LIN {X 0,Y 177.119,Z 453.02,A -85,B 0,C 180,E1 -22409.999,E2 -22409.999} C_VEL
LIN {X 0,Y 176.439,Z 454.874,A -85,B 0,C 180,E1 -22414.569,E2 -22414.569} C_VEL
LIN {X 0,Y 176.286,Z 455.203,A -85,B 0,C 180,E1 -22416.868,E2 -22416.868} C_VEL
LIN {X 0,Y 176.801,Z 454.648,A -85,B 0,C 180,E1 -22421.463,E2 -22421.463} C_VEL
LIN {X 0,Y 178.406,Z 452.583,A -85,B 0,C 180,E1 -22426.006,E2 -22426.006} C_VEL
LIN {X 0,Y 180.457,Z 449.998,A -85,B 0,C 180,E1 -22429.331,E2 -22429.331} C_VEL
LIN {X 0,Y 183.132,Z 446.482,A -85,B 0,C 180,E1 -22432.567,E2 -22432.567} C_VEL
LIN {X 0,Y 186.346,Z 441.993,A -85,B 0,C 180,E1 -22435.703,E2 -22435.703} C_VEL
LIN {X 0,Y 191.105,Z 435.334,A -85,B 0,C 180,E1 -22439.161,E2 -22439.161} C_VEL
LIN {X 0,Y 195.82,Z 428.208,A -85,B 0,C 180,E1 -22441.963,E2 -22441.963} C_VEL
LIN {X 0,Y 201.029,Z 419.477,A -85,B 0,C 180,E1 -22444.617,E2 -22444.617} C_VEL
LIN {X 0,Y 205.808,Z 410.713,A -85,B 0,C 180,E1 -22446.697,E2 -22446.697} C_VEL
LIN {X 0,Y 210.975,Z 400.084,A -85,B 0,C 180,E1 -22448.652,E2 -22448.652} C_VEL
LIN {X 0,Y 215.413,Z 389.657,A -85,B 0,C 180,E1 -22450.117,E2 -22450.117} C_VEL
LIN {X 0,Y 219.48,Z 378.312,A -85,B 0,C 180,E1 -22451.333,E2 -22451.333} C_VEL
LIN {X 0,Y 223.276,Z 364.778,A -85,B 0,C 180,E1 -22452.437,E2 -22452.437} C_VEL
LIN {X 0,Y 226.064,Z 351.459,A -85,B 0,C 180,E1 -22453.198,E2 -22453.198} C_VEL
LIN {X 0,Y 228.603,Z 331.076,A -85,B 0,C 180,E1 -22453.998,E2 -22453.998} C_VEL
LIN {X 0,Y 229.847,Z 318.937,A -85,B 0,C 180,E1 -22454.478,E2 -22454.478} C_VEL
LIN {X 0,Y 229.863,Z 308.216,A -85,B 0,C 180,E1 -22455.412,E2 -22455.412} C_VEL
LIN {X 0,Y 227.63,Z 301.276,A -85,B 0,C 180,E1 -22457.167,E2 -22457.167} C_VEL
LIN {X 0,Y 225.204,Z 295.085,A -85,B 0,C 180,E1 -22459.217,E2 -22459.217} C_VEL
LIN {X 0,Y 223.459,Z 290.853,A -85,B 0,C 180,E1 -22460.87,E2 -22460.87} C_VEL
LIN {X 0,Y 221.449,Z 286.067,A -85,B 0,C 180,E1 -22463.095,E2 -22463.095} C_VEL
LIN {X 0,Y 219.336,Z 281.128,A -85,B 0,C 180,E1 -22466.096,E2 -22466.096} C_VEL
LIN {X 0,Y 217.144,Z 276.417,A -85,B 0,C 180,E1 -22471.174,E2 -22471.174} C_VEL
LIN {X 0,Y 216.832,Z 274.973,A -85,B 0,C 180,E1 -22475.167,E2 -22475.167} C_VEL
LIN {X 0,Y 217.513,Z 275.061,A -85,B 0,C 180,E1 -22478.561,E2 -22478.561} C_VEL
LIN {X 0,Y 218.482,Z 275.796,A -85,B 0,C 180,E1 -22480.742,E2 -22480.742} C_VEL
LIN {X 0,Y 220.281,Z 278.676,A -85,B 0,C 180,E1 -22483.828,E2 -22483.828} C_VEL
LIN {X 0,Y 221.098,Z 279.677,A -85,B 0,C 180,E1 -22484.873,E2 -22484.873} C_VEL
LIN {X 0,Y 223.871,Z 284.056,A -85,B 0,C 180,E1 -22487.867,E2 -22487.867} C_VEL
LIN {X 0,Y 226.551,Z 288.873,A -85,B 0,C 180,E1 -22490.248,E2 -22490.248} C_VEL
LIN {X 0,Y 229.149,Z 293.131,A -85,B 0,C 180,E1 -22492.167,E2 -22492.167} C_VEL
LIN {X 0,Y 231.689,Z 298.864,A -85,B 0,C 180,E1 -22493.945,E2 -22493.945} C_VEL
LIN {X 0,Y 227.767,Z 334.024,A -85,B 0,C 180,E1 -22495.35,E2 -22495.35} C_VEL
LIN {X 0,Y 225.731,Z 345.822,A -85,B 0,C 180,E1 -22496.11,E2 -22496.11} C_VEL
LIN {X 0,Y 222.631,Z 358.855,A -85,B 0,C 180,E1 -22497.286,E2 -22497.286} C_VEL
LIN {X 0,Y 218.74,Z 371.166,A -85,B 0,C 180,E1 -22498.758,E2 -22498.758} C_VEL
LIN {X 0,Y 214.991,Z 380.89,A -85,B 0,C 180,E1 -22500.234,E2 -22500.234} C_VEL
LIN {X 0,Y 210.962,Z 389.896,A -85,B 0,C 180,E1 -22501.957,E2 -22501.957} C_VEL
LIN {X 0,Y 205.904,Z 399.515,A -85,B 0,C 180,E1 -22504.288,E2 -22504.288} C_VEL
LIN {X 0,Y 200.682,Z 408.153,A -85,B 0,C 180,E1 -22507.04,E2 -22507.04} C_VEL
LIN {X 0,Y 196.113,Z 414.843,A -85,B 0,C 180,E1 -22509.8,E2 -22509.8} C_VEL
LIN {X 0,Y 192.012,Z 420.181,A -85,B 0,C 180,E1 -22512.686,E2 -22512.686} C_VEL
LIN {X 0,Y 187.629,Z 425.077,A -85,B 0,C 180,E1 -22516.315,E2 -22516.315} C_VEL
LIN {X 0,Y 183.961,Z 428.518,A -85,B 0,C 180,E1 -22520.11,E2 -22520.11} C_VEL
LIN {X 0,Y 181.959,Z 430.045,A -85,B 0,C 180,E1 -22522.721,E2 -22522.721} C_VEL
LIN {X 0,Y 179.89,Z 431.131,A -85,B 0,C 180,E1 -22526.03,E2 -22526.03} C_VEL
LIN {X 0,Y 178.152,Z 431.262,A -85,B 0,C 180,E1 -22529.787,E2 -22529.787} C_VEL
LIN {X 0,Y 176.979,Z 430.196,A -85,B 0,C 180,E1 -22533.776,E2 -22533.776} C_VEL
LIN {X 0,Y 176.467,Z 428.319,A -85,B 0,C 180,E1 -22537.201,E2 -22537.201} C_VEL
LIN {X 0,Y 176.435,Z 425.306,A -85,B 0,C 180,E1 -22540.815,E2 -22540.815} C_VEL
LIN {X 0,Y 176.901,Z 421.239,A -85,B 0,C 180,E1 -22544.349,E2 -22544.349} C_VEL
LIN {X 0,Y 177.667,Z 416.16,A -85,B 0,C 180,E1 -22547.743,E2 -22547.743} C_VEL
LIN {X 0,Y 178.652,Z 410.046,A -85,B 0,C 180,E1 -22550.993,E2 -22550.993} C_VEL
LIN {X 0,Y 180.024,Z 402.659,A -85,B 0,C 180,E1 -22554.156,E2 -22554.156} C_VEL
LIN {X 0,Y 181.84,Z 393.663,A -85,B 0,C 180,E1 -22557.243,E2 -22557.243} C_VEL
LIN {X 0,Y 183.867,Z 382.77,A -85,B 0,C 180,E1 -22560.205,E2 -22560.205} C_VEL
LIN {X 0,Y 185.651,Z 372.786,A -85,B 0,C 180,E1 -22562.372,E2 -22562.372} C_VEL
LIN {X 0,Y 187.482,Z 361.225,A -85,B 0,C 180,E1 -22564.361,E2 -22564.361} C_VEL
LIN {X 0,Y 189.182,Z 348.375,A -85,B 0,C 180,E1 -22566.059,E2 -22566.059} C_VEL
LIN {X 0,Y 190.453,Z 335.541,A -85,B 0,C 180,E1 -22567.3,E2 -22567.3} C_VEL
LIN {X 0,Y 191.289,Z 323.154,A -85,B 0,C 180,E1 -22568.117,E2 -22568.117} C_VEL
LIN {X 0,Y 194.053,Z 269.424,A -85,B 0,C 180,E1 -22570.531,E2 -22570.531} C_VEL
LIN {X 0,Y 183.64,Z 244.117,A -85,B 0,C 180,E1 -22573.175,E2 -22573.175} C_VEL
LIN {X 0,Y 178.833,Z 233.185,A -85,B 0,C 180,E1 -22574.472,E2 -22574.472} C_VEL
LIN {X 0,Y 178.665,Z 232.231,A -85,B 0,C 180,E1 -22574.603,E2 -22574.603} C_VEL
LIN {X 0,Y 178.836,Z 232.21,A -85,B 0,C 180,E1 -22579.254,E2 -22579.254} C_VEL
LIN {X 0,Y 178.901,Z 232.2,A -85,B 0,C 180,E1 -22583.232,E2 -22583.232} C_VEL
LIN {X 0,Y 179.148,Z 232.168,A -85,B 0,C 180,E1 -22587.752,E2 -22587.752} C_VEL
LIN {X 0,Y 179.366,Z 232.141,A -85,B 0,C 180,E1 -22590.001,E2 -22590.001} C_VEL
LIN {X 0,Y 178.853,Z 232.206,A -85,B 0,C 180,E1 -22594.508,E2 -22594.508} C_VEL
LIN {X 0,Y 178.909,Z 232.197,A -85,B 0,C 180,E1 -22599.041,E2 -22599.041} C_VEL
LIN {X 0,Y 178.659,Z 232.23,A -85,B 0,C 180,E1 -22603.653,E2 -22603.653} C_VEL
LIN {X 0,Y 178.624,Z 232.228,A -85,B 0,C 180,E1 -22609.216,E2 -22609.216} C_VEL
LIN {X 0,Y 178.517,Z 232.241,A -85,B 0,C 180,E1 -22615.112,E2 -22615.112} C_VEL
LIN {X 0,Y 178.461,Z 232.253,A -85,B 0,C 180,E1 -22620.795,E2 -22620.795} C_VEL
LIN {X 0,Y 178.484,Z 232.239,A -85,B 0,C 180,E1 -22624.219,E2 -22624.219} C_VEL
LIN {X 0,Y 178.389,Z 232.236,A -85,B 0,C 180,E1 -22629.077,E2 -22629.077} C_VEL
LIN {X 0,Y 178.396,Z 232.253,A -85,B 0,C 180,E1 -22632.047,E2 -22632.047} C_VEL
LIN {X 0,Y 178.394,Z 232.26,A -85,B 0,C 180,E1 -22635.165,E2 -22635.165} C_VEL
LIN {X 0,Y 178.401,Z 232.261,A -85,B 0,C 180,E1 -22638.461,E2 -22638.461} C_VEL
LIN {X 0,Y 178.422,Z 232.253,A -85,B 0,C 180,E1 -22643.783,E2 -22643.783} C_VEL
LIN {X 0,Y 178.486,Z 232.249,A -85,B 0,C 180,E1 -22646.547,E2 -22646.547} C_VEL
LIN {X 0,Y 178.446,Z 232.252,A -85,B 0,C 180,E1 -22651.796,E2 -22651.796} C_VEL
LIN {X 0,Y 178.518,Z 232.239,A -85,B 0,C 180,E1 -22654.889,E2 -22654.889} C_VEL
LIN {X 0,Y 178.623,Z 232.235,A -85,B 0,C 180,E1 -22660.787,E2 -22660.787} C_VEL
LIN {X 0,Y 178.652,Z 232.216,A -85,B 0,C 180,E1 -22666.348,E2 -22666.348} C_VEL
LIN {X 0,Y 178.907,Z 232.168,A -85,B 0,C 180,E1 -22670.96,E2 -22670.96} C_VEL
LIN {X 0,Y 179.146,Z 232.166,A -85,B 0,C 180,E1 -22677.752,E2 -22677.752} C_VEL
LIN {X 0,Y 179.349,Z 232.144,A -85,B 0,C 180,E1 -22680,E2 -22680} C_VEL
LIN {X 0,Y 178.839,Z 232.199,A -85,B 0,C 180,E1 -22684.508,E2 -22684.508} C_VEL
LIN {X 0,Y 178.909,Z 232.183,A -85,B 0,C 180,E1 -22689.041,E2 -22689.041} C_VEL
LIN {X 0,Y 178.645,Z 232.232,A -85,B 0,C 180,E1 -22693.653,E2 -22693.653} C_VEL
LIN {X 0,Y 178.559,Z 232.238,A -85,B 0,C 180,E1 -22699.154,E2 -22699.154} C_VEL
LIN {X 0,Y 178.507,Z 232.25,A -85,B 0,C 180,E1 -22705.103,E2 -22705.103} C_VEL
LIN {X 0,Y 178.463,Z 232.246,A -85,B 0,C 180,E1 -22710.794,E2 -22710.794} C_VEL
LIN {X 0,Y 178.485,Z 232.251,A -85,B 0,C 180,E1 -22714.218,E2 -22714.218} C_VEL
LIN {X 0,Y 178.389,Z 232.267,A -85,B 0,C 180,E1 -22719.076,E2 -22719.076} C_VEL
LIN {X 0,Y 178.395,Z 232.266,A -85,B 0,C 180,E1 -22722.046,E2 -22722.046} C_VEL
LIN {X 0,Y 178.444,Z 232.289,A -85,B 0,C 180,E1 -22727.474,E2 -22727.474} C_VEL
LIN {X 0,Y 180.599,Z 241.672,A -85,B 0,C 180,E1 -22732,E2 -22732} C_VEL
LIN {X 0,Y 181.124,Z 244.073,A -85,B 0,C 180,E1 -22733.042,E2 -22733.042} C_VEL
LIN {X 0,Y 188.923,Z 267.082,A -85,B 0,C 180,E1 -22735.312,E2 -22735.312} C_VEL
LIN {X 0,Y 192.659,Z 311.704,A -85,B 0,C 180,E1 -22738.04,E2 -22738.04} C_VEL
LIN {X 0,Y 190.324,Z 354.639,A -85,B 0,C 180,E1 -22740.022,E2 -22740.022} C_VEL
LIN {X 0,Y 189.127,Z 367.936,A -85,B 0,C 180,E1 -22741.036,E2 -22741.036} C_VEL
LIN {X 0,Y 187.45,Z 380.188,A -85,B 0,C 180,E1 -22742.356,E2 -22742.356} C_VEL
LIN {X 0,Y 187.163,Z 381.965,A -85,B 0,C 180,E1 -22742.59,E2 -22742.59} C_VEL
LIN {X 0,Y 185.633,Z 387.249,A -85,B 0,C 180,E1 -22743.275,E2 -22743.275} C_VEL
LIN {X 0,Y 181.389,Z 395.413,A -85,B 0,C 180,E1 -22744.432,E2 -22744.432} C_VEL
LIN {X 0,Y 177.063,Z 403.193,A -85,B 0,C 180,E1 -22745.844,E2 -22745.844} C_VEL
LIN {X 0,Y 175.47,Z 407.827,A -85,B 0,C 180,E1 -22746.925,E2 -22746.925} C_VEL
LIN {X 0,Y 173.738,Z 416.402,A -85,B 0,C 180,E1 -22749.27,E2 -22749.27} C_VEL
LIN {X 0,Y 172.106,Z 424.998,A -85,B 0,C 180,E1 -22752.165,E2 -22752.165} C_VEL
LIN {X 0,Y 170.744,Z 433.367,A -85,B 0,C 180,E1 -22755.701,E2 -22755.701} C_VEL
LIN {X 0,Y 169.897,Z 440.053,A -85,B 0,C 180,E1 -22759.271,E2 -22759.271} C_VEL
LIN {X 0,Y 169.659,Z 445.327,A -85,B 0,C 180,E1 -22762.861,E2 -22762.861} C_VEL
LIN {X 0,Y 169.695,Z 449.31,A -85,B 0,C 180,E1 -22766.438,E2 -22766.438} C_VEL
LIN {X 0,Y 170.06,Z 452.158,A -85,B 0,C 180,E1 -22769.999,E2 -22769.999} C_VEL
LIN {X 0,Y 169.559,Z 453.36,A -85,B 0,C 180,E1 -22772.375,E2 -22772.375} C_VEL
LIN {X 0,Y 169.309,Z 454.199,A -85,B 0,C 180,E1 -22774.969,E2 -22774.969} C_VEL
LIN {X 0,Y 169.382,Z 454.571,A -85,B 0,C 180,E1 -22779.553,E2 -22779.553} C_VEL
LIN {X 0,Y 169.809,Z 454.212,A -85,B 0,C 180,E1 -22781.942,E2 -22781.942} C_VEL
LIN {X 0,Y 170.468,Z 453.443,A -85,B 0,C 180,E1 -22784.321,E2 -22784.321} C_VEL
LIN {X 0,Y 172.966,Z 450.792,A -85,B 0,C 180,E1 -22788.968,E2 -22788.968} C_VEL
LIN {X 0,Y 175.597,Z 447.772,A -85,B 0,C 180,E1 -22792.347,E2 -22792.347} C_VEL
LIN {X 0,Y 178.737,Z 443.798,A -85,B 0,C 180,E1 -22795.627,E2 -22795.627} C_VEL
LIN {X 0,Y 182.693,Z 438.765,A -85,B 0,C 180,E1 -22798.741,E2 -22798.741} C_VEL
LIN {X 0,Y 188.219,Z 431.419,A -85,B 0,C 180,E1 -22802.146,E2 -22802.146} C_VEL
LIN {X 0,Y 193.406,Z 423.633,A -85,B 0,C 180,E1 -22804.912,E2 -22804.912} C_VEL
LIN {X 0,Y 199.229,Z 414.009,A -85,B 0,C 180,E1 -22807.481,E2 -22807.481} C_VEL
LIN {X 0,Y 205.063,Z 403.155,A -85,B 0,C 180,E1 -22809.666,E2 -22809.666} C_VEL
LIN {X 0,Y 210.125,Z 392.195,A -85,B 0,C 180,E1 -22811.343,E2 -22811.343} C_VEL
LIN {X 0,Y 214.917,Z 380.063,A -85,B 0,C 180,E1 -22812.73,E2 -22812.73} C_VEL
LIN {X 0,Y 218.864,Z 367.436,A -85,B 0,C 180,E1 -22813.82,E2 -22813.82} C_VEL
LIN {X 0,Y 222.233,Z 353.055,A -85,B 0,C 180,E1 -22814.684,E2 -22814.684} C_VEL
LIN {X 0,Y 224.374,Z 338.166,A -85,B 0,C 180,E1 -22815.313,E2 -22815.313} C_VEL
LIN {X 0,Y 226.349,Z 320.431,A -85,B 0,C 180,E1 -22815.981,E2 -22815.981} C_VEL
LIN {X 0,Y 226.445,Z 311.706,A -85,B 0,C 180,E1 -22816.757,E2 -22816.757} C_VEL
LIN {X 0,Y 224.476,Z 305.423,A -85,B 0,C 180,E1 -22818.521,E2 -22818.521} C_VEL
LIN {X 0,Y 222.16,Z 299.016,A -85,B 0,C 180,E1 -22820.75,E2 -22820.75} C_VEL
LIN {X 0,Y 219.477,Z 292.206,A -85,B 0,C 180,E1 -22823.873,E2 -22823.873} C_VEL
LIN {X 0,Y 217.606,Z 287.533,A -85,B 0,C 180,E1 -22826.839,E2 -22826.839} C_VEL
LIN {X 0,Y 215.872,Z 283.278,A -85,B 0,C 180,E1 -22831.523,E2 -22831.523} C_VEL
LIN {X 0,Y 215.606,Z 282.016,A -85,B 0,C 180,E1 -22834.928,E2 -22834.928} C_VEL
LIN {X 0,Y 216.237,Z 282.017,A -85,B 0,C 180,E1 -22838.308,E2 -22838.308} C_VEL
LIN {X 0,Y 217.131,Z 282.762,A -85,B 0,C 180,E1 -22840.482,E2 -22840.482} C_VEL
LIN {X 0,Y 218.962,Z 285.684,A -85,B 0,C 180,E1 -22843.728,E2 -22843.728} C_VEL
LIN {X 0,Y 219.724,Z 286.945,A -85,B 0,C 180,E1 -22844.777,E2 -22844.777} C_VEL
LIN {X 0,Y 221.955,Z 290.54,A -85,B 0,C 180,E1 -22847.296,E2 -22847.296} C_VEL
LIN {X 0,Y 225.952,Z 297.719,A -85,B 0,C 180,E1 -22850.854,E2 -22850.854} C_VEL
LIN {X 0,Y 227.994,Z 302.296,A -85,B 0,C 180,E1 -22852.465,E2 -22852.465} C_VEL
LIN {X 0,Y 227.921,Z 303.854,A -85,B 0,C 180,E1 -22852.582,E2 -22852.582} C_VEL
LIN {X 0,Y 224.199,Z 334.973,A -85,B 0,C 180,E1 -22853.813,E2 -22853.813} C_VEL
LIN {X 0,Y 221.768,Z 348.22,A -85,B 0,C 180,E1 -22854.691,E2 -22854.691} C_VEL
LIN {X 0,Y 218.432,Z 360.975,A -85,B 0,C 180,E1 -22855.877,E2 -22855.877} C_VEL
LIN {X 0,Y 214.802,Z 371.788,A -85,B 0,C 180,E1 -22857.187,E2 -22857.187} C_VEL
LIN {X 0,Y 210.261,Z 382.84,A -85,B 0,C 180,E1 -22858.9,E2 -22858.9} C_VEL
LIN {X 0,Y 205.124,Z 393.271,A -85,B 0,C 180,E1 -22861.023,E2 -22861.023} C_VEL
LIN {X 0,Y 200.669,Z 401.09,A -85,B 0,C 180,E1 -22863.011,E2 -22863.011} C_VEL
LIN {X 0,Y 195.312,Z 409.43,A -85,B 0,C 180,E1 -22865.75,E2 -22865.75} C_VEL
LIN {X 0,Y 190.607,Z 415.793,A -85,B 0,C 180,E1 -22868.481,E2 -22868.481} C_VEL
LIN {X 0,Y 186.35,Z 420.875,A -85,B 0,C 180,E1 -22871.317,E2 -22871.317} C_VEL
LIN {X 0,Y 181.81,Z 425.611,A -85,B 0,C 180,E1 -22874.899,E2 -22874.899} C_VEL
LIN {X 0,Y 178.003,Z 428.956,A -85,B 0,C 180,E1 -22878.636,E2 -22878.636} C_VEL
LIN {X 0,Y 174.915,Z 431.015,A -85,B 0,C 180,E1 -22882.464,E2 -22882.464} C_VEL
LIN {X 0,Y 172.403,Z 431.917,A -85,B 0,C 180,E1 -22886.642,E2 -22886.642} C_VEL
LIN {X 0,Y 170.871,Z 431.64,A -85,B 0,C 180,E1 -22890.262,E2 -22890.262} C_VEL
LIN {X 0,Y 169.802,Z 430.318,A -85,B 0,C 180,E1 -22894.129,E2 -22894.129} C_VEL
LIN {X 0,Y 169.288,Z 427.501,A -85,B 0,C 180,E1 -22898.515,E2 -22898.515} C_VEL
LIN {X 0,Y 169.583,Z 422.962,A -85,B 0,C 180,E1 -22903.14,E2 -22903.14} C_VEL
LIN {X 0,Y 170.389,Z 417.424,A -85,B 0,C 180,E1 -22907.197,E2 -22907.197} C_VEL
LIN {X 0,Y 171.358,Z 411.646,A -85,B 0,C 180,E1 -22910.499,E2 -22910.499} C_VEL
LIN {X 0,Y 172.763,Z 404.104,A -85,B 0,C 180,E1 -22913.947,E2 -22913.947} C_VEL
LIN {X 0,Y 174.568,Z 395.284,A -85,B 0,C 180,E1 -22917.178,E2 -22917.178} C_VEL
LIN {X 0,Y 176.473,Z 385.292,A -85,B 0,C 180,E1 -22920.097,E2 -22920.097} C_VEL
LIN {X 0,Y 178.548,Z 374.345,A -85,B 0,C 180,E1 -22922.633,E2 -22922.633} C_VEL
LIN {X 0,Y 180.465,Z 362.571,A -85,B 0,C 180,E1 -22924.785,E2 -22924.785} C_VEL
LIN {X 0,Y 182.199,Z 350.177,A -85,B 0,C 180,E1 -22926.512,E2 -22926.512} C_VEL
LIN {X 0,Y 183.651,Z 336.993,A -85,B 0,C 180,E1 -22927.871,E2 -22927.871} C_VEL
LIN {X 0,Y 184.478,Z 324.654,A -85,B 0,C 180,E1 -22928.746,E2 -22928.746} C_VEL
LIN {X 0,Y 187.377,Z 270.971,A -85,B 0,C 180,E1 -22931.245,E2 -22931.245} C_VEL
LIN {X 0,Y 176.862,Z 245.4,A -85,B 0,C 180,E1 -22934.074,E2 -22934.074} C_VEL
LIN {X 0,Y 171.755,Z 233.904,A -85,B 0,C 180,E1 -22935.516,E2 -22935.516} C_VEL
LIN {X 0,Y 171.601,Z 233.11,A -85,B 0,C 180,E1 -22935.639,E2 -22935.639} C_VEL
LIN {X 0,Y 171.845,Z 233.081,A -85,B 0,C 180,E1 -22940.585,E2 -22940.585} C_VEL
LIN {X 0,Y 171.806,Z 233.083,A -85,B 0,C 180,E1 -22945.308,E2 -22945.308} C_VEL
LIN {X 0,Y 172.329,Z 233.018,A -85,B 0,C 180,E1 -22950.001,E2 -22950.001} C_VEL
LIN {X 0,Y 171.802,Z 233.084,A -85,B 0,C 180,E1 -22954.694,E2 -22954.694} C_VEL
LIN {X 0,Y 171.847,Z 233.077,A -85,B 0,C 180,E1 -22959.416,E2 -22959.416} C_VEL
LIN {X 0,Y 171.578,Z 233.113,A -85,B 0,C 180,E1 -22964.228,E2 -22964.228} C_VEL
LIN {X 0,Y 171.543,Z 233.108,A -85,B 0,C 180,E1 -22969.56,E2 -22969.56} C_VEL
LIN {X 0,Y 171.445,Z 233.124,A -85,B 0,C 180,E1 -22975.599,E2 -22975.599} C_VEL
LIN {X 0,Y 171.419,Z 233.13,A -85,B 0,C 180,E1 -22980.573,E2 -22980.573} C_VEL
LIN {X 0,Y 171.393,Z 233.118,A -85,B 0,C 180,E1 -22985.036,E2 -22985.036} C_VEL
LIN {X 0,Y 171.345,Z 233.112,A -85,B 0,C 180,E1 -22988.802,E2 -22988.802} C_VEL
LIN {X 0,Y 171.321,Z 233.14,A -85,B 0,C 180,E1 -22994.218,E2 -22994.218} C_VEL
LIN {X 0,Y 171.333,Z 233.143,A -85,B 0,C 180,E1 -22998.981,E2 -22998.981} C_VEL
LIN {X 0,Y 171.363,Z 233.131,A -85,B 0,C 180,E1 -23002.035,E2 -23002.035} C_VEL
LIN {X 0,Y 171.399,Z 233.129,A -85,B 0,C 180,E1 -23005.093,E2 -23005.093} C_VEL
LIN {X 0,Y 171.411,Z 233.132,A -85,B 0,C 180,E1 -23010.527,E2 -23010.527} C_VEL
LIN {X 0,Y 171.443,Z 233.122,A -85,B 0,C 180,E1 -23015.8,E2 -23015.8} C_VEL
LIN {X 0,Y 171.579,Z 233.112,A -85,B 0,C 180,E1 -23020.872,E2 -23020.872} C_VEL
LIN {X 0,Y 171.569,Z 233.1,A -85,B 0,C 180,E1 -23025.772,E2 -23025.772} C_VEL
LIN {X 0,Y 171.846,Z 233.044,A -85,B 0,C 180,E1 -23030.585,E2 -23030.585} C_VEL
LIN {X 0,Y 171.801,Z 233.076,A -85,B 0,C 180,E1 -23035.307,E2 -23035.307} C_VEL
LIN {X 0,Y 172.314,Z 233.021,A -85,B 0,C 180,E1 -23040,E2 -23040} C_VEL
LIN {X 0,Y 171.789,Z 233.076,A -85,B 0,C 180,E1 -23044.693,E2 -23044.693} C_VEL
LIN {X 0,Y 171.847,Z 233.062,A -85,B 0,C 180,E1 -23049.415,E2 -23049.415} C_VEL
LIN {X 0,Y 171.56,Z 233.118,A -85,B 0,C 180,E1 -23054.229,E2 -23054.229} C_VEL
LIN {X 0,Y 171.485,Z 233.117,A -85,B 0,C 180,E1 -23059.502,E2 -23059.502} C_VEL
LIN {X 0,Y 171.438,Z 233.133,A -85,B 0,C 180,E1 -23065.592,E2 -23065.592} C_VEL
LIN {X 0,Y 171.42,Z 233.123,A -85,B 0,C 180,E1 -23070.572,E2 -23070.572} C_VEL
LIN {X 0,Y 171.394,Z 233.135,A -85,B 0,C 180,E1 -23075.035,E2 -23075.035} C_VEL
LIN {X 0,Y 171.345,Z 233.144,A -85,B 0,C 180,E1 -23078.801,E2 -23078.801} C_VEL
LIN {X 0,Y 171.32,Z 233.147,A -85,B 0,C 180,E1 -23084.218,E2 -23084.218} C_VEL
LIN {X 0,Y 171.369,Z 233.182,A -85,B 0,C 180,E1 -23086.824,E2 -23086.824} C_VEL
LIN {X 0,Y 173.685,Z 243.165,A -85,B 0,C 180,E1 -23091.833,E2 -23091.833} C_VEL
LIN {X 0,Y 181.918,Z 267.185,A -85,B 0,C 180,E1 -23094.424,E2 -23094.424} C_VEL
LIN {X 0,Y 182.53,Z 270.033,A -85,B 0,C 180,E1 -23094.659,E2 -23094.659} C_VEL
LIN {X 0,Y 185.969,Z 312.533,A -85,B 0,C 180,E1 -23097.34,E2 -23097.34} C_VEL
LIN {X 0,Y 183.579,Z 354.446,A -85,B 0,C 180,E1 -23099.359,E2 -23099.359} C_VEL
LIN {X 0,Y 182.344,Z 367.607,A -85,B 0,C 180,E1 -23100.407,E2 -23100.407} C_VEL
LIN {X 0,Y 180.547,Z 380.248,A -85,B 0,C 180,E1 -23101.836,E2 -23101.836} C_VEL
LIN {X 0,Y 178.489,Z 392.416,A -85,B 0,C 180,E1 -23103.706,E2 -23103.706} C_VEL
LIN {X 0,Y 176.39,Z 403.457,A -85,B 0,C 180,E1 -23105.895,E2 -23105.895} C_VEL
LIN {X 0,Y 175.47,Z 407.827,A -85,B 0,C 180,E1 -23106.925,E2 -23106.925} C_VEL
LIN {X 0,Y 173.907,Z 412.344,A -85,B 0,C 180,E1 -23108.079,E2 -23108.079} C_VEL
LIN {X 0,Y 169.671,Z 419.094,A -85,B 0,C 180,E1 -23110.053,E2 -23110.053} C_VEL
LIN {X 0,Y 165.572,Z 425.352,A -85,B 0,C 180,E1 -23112.283,E2 -23112.283} C_VEL
LIN {X 0,Y 164.241,Z 429.003,A -85,B 0,C 180,E1 -23113.828,E2 -23113.828} C_VEL
LIN {X 0,Y 163.117,Z 436.508,A -85,B 0,C 180,E1 -23117.559,E2 -23117.559} C_VEL
LIN {X 0,Y 162.645,Z 442.441,A -85,B 0,C 180,E1 -23121.301,E2 -23121.301} C_VEL
LIN {X 0,Y 162.661,Z 447.013,A -85,B 0,C 180,E1 -23125.042,E2 -23125.042} C_VEL
LIN {X 0,Y 162.67,Z 449.333,A -85,B 0,C 180,E1 -23127.523,E2 -23127.523} C_VEL
LIN {X 0,Y 163.001,Z 451.213,A -85,B 0,C 180,E1 -23129.999,E2 -23129.999} C_VEL
LIN {X 0,Y 162.494,Z 452.526,A -85,B 0,C 180,E1 -23132.478,E2 -23132.478} C_VEL
LIN {X 0,Y 162.255,Z 453.418,A -85,B 0,C 180,E1 -23134.969,E2 -23134.969} C_VEL
LIN {X 0,Y 162.35,Z 453.989,A -85,B 0,C 180,E1 -23139.971,E2 -23139.971} C_VEL
LIN {X 0,Y 163.559,Z 453.071,A -85,B 0,C 180,E1 -23144.94,E2 -23144.94} C_VEL
LIN {X 0,Y 166.227,Z 450.623,A -85,B 0,C 180,E1 -23149.769,E2 -23149.769} C_VEL
LIN {X 0,Y 170.018,Z 446.61,A -85,B 0,C 180,E1 -23154.416,E2 -23154.416} C_VEL
LIN {X 0,Y 173.66,Z 442.488,A -85,B 0,C 180,E1 -23157.736,E2 -23157.736} C_VEL
LIN {X 0,Y 178.08,Z 437.328,A -85,B 0,C 180,E1 -23160.867,E2 -23160.867} C_VEL
LIN {X 0,Y 183.143,Z 430.965,A -85,B 0,C 180,E1 -23163.809,E2 -23163.809} C_VEL
LIN {X 0,Y 188.704,Z 423.196,A -85,B 0,C 180,E1 -23166.576,E2 -23166.576} C_VEL
LIN {X 0,Y 194.786,Z 413.681,A -85,B 0,C 180,E1 -23169.154,E2 -23169.154} C_VEL
LIN {X 0,Y 200.87,Z 402.987,A -85,B 0,C 180,E1 -23171.329,E2 -23171.329} C_VEL
LIN {X 0,Y 206.164,Z 392.16,A -85,B 0,C 180,E1 -23172.983,E2 -23172.983} C_VEL
LIN {X 0,Y 211.124,Z 380.135,A -85,B 0,C 180,E1 -23174.351,E2 -23174.351} C_VEL
LIN {X 0,Y 215.206,Z 367.755,A -85,B 0,C 180,E1 -23175.425,E2 -23175.425} C_VEL
LIN {X 0,Y 218.892,Z 352.781,A -85,B 0,C 180,E1 -23176.329,E2 -23176.329} C_VEL
LIN {X 0,Y 221.095,Z 338.721,A -85,B 0,C 180,E1 -23176.926,E2 -23176.926} C_VEL
LIN {X 0,Y 223.132,Z 321.348,A -85,B 0,C 180,E1 -23177.592,E2 -23177.592} C_VEL
LIN {X 0,Y 223.248,Z 315.345,A -85,B 0,C 180,E1 -23178.164,E2 -23178.164} C_VEL
LIN {X 0,Y 221.261,Z 308.893,A -85,B 0,C 180,E1 -23180.118,E2 -23180.118} C_VEL
LIN {X 0,Y 219.262,Z 303.07,A -85,B 0,C 180,E1 -23182.409,E2 -23182.409} C_VEL
LIN {X 0,Y 217.739,Z 298.684,A -85,B 0,C 180,E1 -23184.48,E2 -23184.48} C_VEL
LIN {X 0,Y 215.982,Z 294.038,A -85,B 0,C 180,E1 -23187.505,E2 -23187.505} C_VEL
LIN {X 0,Y 214.607,Z 290.162,A -85,B 0,C 180,E1 -23191.869,E2 -23191.869} C_VEL
LIN {X 0,Y 214.394,Z 289.062,A -85,B 0,C 180,E1 -23194.776,E2 -23194.776} C_VEL
LIN {X 0,Y 214.901,Z 288.939,A -85,B 0,C 180,E1 -23197.78,E2 -23197.78} C_VEL
LIN {X 0,Y 215.764,Z 289.598,A -85,B 0,C 180,E1 -23200.142,E2 -23200.142} C_VEL
LIN {X 0,Y 217.569,Z 292.585,A -85,B 0,C 180,E1 -23203.521,E2 -23203.521} C_VEL
LIN {X 0,Y 220.054,Z 297.03,A -85,B 0,C 180,E1 -23206.712,E2 -23206.712} C_VEL
LIN {X 0,Y 223.937,Z 304.441,A -85,B 0,C 180,E1 -23210.397,E2 -23210.397} C_VEL
LIN {X 0,Y 224.667,Z 306.055,A -85,B 0,C 180,E1 -23211.001,E2 -23211.001} C_VEL
LIN {X 0,Y 220.975,Z 335.59,A -85,B 0,C 180,E1 -23212.194,E2 -23212.194} C_VEL
LIN {X 0,Y 218.385,Z 348.849,A -85,B 0,C 180,E1 -23213.068,E2 -23213.068} C_VEL
LIN {X 0,Y 214.878,Z 361.548,A -85,B 0,C 180,E1 -23214.251,E2 -23214.251} C_VEL
LIN {X 0,Y 210.96,Z 372.706,A -85,B 0,C 180,E1 -23215.6,E2 -23215.6} C_VEL
LIN {X 0,Y 206.793,Z 382.436,A -85,B 0,C 180,E1 -23217.078,E2 -23217.078} C_VEL
LIN {X 0,Y 201.859,Z 392.27,A -85,B 0,C 180,E1 -23219.001,E2 -23219.001} C_VEL
LIN {X 0,Y 196.058,Z 401.957,A -85,B 0,C 180,E1 -23221.45,E2 -23221.45} C_VEL
LIN {X 0,Y 190.277,Z 410.34,A -85,B 0,C 180,E1 -23224.248,E2 -23224.248} C_VEL
LIN {X 0,Y 184.341,Z 417.751,A -85,B 0,C 180,E1 -23227.588,E2 -23227.588} C_VEL
LIN {X 0,Y 178.803,Z 423.722,A -85,B 0,C 180,E1 -23231.334,E2 -23231.334} C_VEL
LIN {X 0,Y 174.479,Z 427.602,A -85,B 0,C 180,E1 -23234.826,E2 -23234.826} C_VEL
LIN {X 0,Y 170.098,Z 430.771,A -85,B 0,C 180,E1 -23239.301,E2 -23239.301} C_VEL
LIN {X 0,Y 167.558,Z 432.046,A -85,B 0,C 180,E1 -23242.669,E2 -23242.669} C_VEL
LIN {X 0,Y 165.197,Z 432.501,A -85,B 0,C 180,E1 -23246.697,E2 -23246.697} C_VEL
LIN {X 0,Y 163.469,Z 431.772,A -85,B 0,C 180,E1 -23251.058,E2 -23251.058} C_VEL
LIN {X 0,Y 162.571,Z 430.162,A -85,B 0,C 180,E1 -23254.778,E2 -23254.778} C_VEL
LIN {X 0,Y 162.186,Z 427.442,A -85,B 0,C 180,E1 -23258.741,E2 -23258.741} C_VEL
LIN {X 0,Y 162.399,Z 423.68,A -85,B 0,C 180,E1 -23262.635,E2 -23262.635} C_VEL
LIN {X 0,Y 163.109,Z 418.859,A -85,B 0,C 180,E1 -23266.418,E2 -23266.418} C_VEL
LIN {X 0,Y 164.187,Z 412.33,A -85,B 0,C 180,E1 -23270.398,E2 -23270.398} C_VEL
LIN {X 0,Y 165.52,Z 405.342,A -85,B 0,C 180,E1 -23273.779,E2 -23273.779} C_VEL
LIN {X 0,Y 167.308,Z 396.678,A -85,B 0,C 180,E1 -23277.154,E2 -23277.154} C_VEL
LIN {X 0,Y 169.225,Z 387.261,A -85,B 0,C 180,E1 -23280.109,E2 -23280.109} C_VEL
LIN {X 0,Y 171.409,Z 376.141,A -85,B 0,C 180,E1 -23282.862,E2 -23282.862} C_VEL
LIN {X 0,Y 173.365,Z 364.542,A -85,B 0,C 180,E1 -23285.129,E2 -23285.129} C_VEL
LIN {X 0,Y 175.165,Z 352.658,A -85,B 0,C 180,E1 -23286.914,E2 -23286.914} C_VEL
LIN {X 0,Y 176.792,Z 338.632,A -85,B 0,C 180,E1 -23288.464,E2 -23288.464} C_VEL
LIN {X 0,Y 177.757,Z 325.449,A -85,B 0,C 180,E1 -23289.459,E2 -23289.459} C_VEL
LIN {X 0,Y 180.813,Z 272.917,A -85,B 0,C 180,E1 -23291.982,E2 -23291.982} C_VEL
LIN {X 0,Y 171.497,Z 250.026,A -85,B 0,C 180,E1 -23294.601,E2 -23294.601} C_VEL
LIN {X 0,Y 164.759,Z 234.975,A -85,B 0,C 180,E1 -23296.59,E2 -23296.59} C_VEL
LIN {X 0,Y 164.563,Z 233.988,A -85,B 0,C 180,E1 -23296.731,E2 -23296.731} C_VEL
LIN {X 0,Y 164.771,Z 233.962,A -85,B 0,C 180,E1 -23300.177,E2 -23300.177} C_VEL
LIN {X 0,Y 164.824,Z 233.955,A -85,B 0,C 180,E1 -23302.651,E2 -23302.651} C_VEL
LIN {X 0,Y 165.043,Z 233.925,A -85,B 0,C 180,E1 -23307.56,E2 -23307.56} C_VEL
LIN {X 0,Y 165.291,Z 233.894,A -85,B 0,C 180,E1 -23310.001,E2 -23310.001} C_VEL
LIN {X 0,Y 164.751,Z 233.961,A -85,B 0,C 180,E1 -23314.895,E2 -23314.895} C_VEL
LIN {X 0,Y 164.826,Z 233.951,A -85,B 0,C 180,E1 -23317.35,E2 -23317.35} C_VEL
LIN {X 0,Y 164.704,Z 233.967,A -85,B 0,C 180,E1 -23321.061,E2 -23321.061} C_VEL
LIN {X 0,Y 164.485,Z 233.994,A -85,B 0,C 180,E1 -23327.404,E2 -23327.404} C_VEL
LIN {X 0,Y 164.474,Z 233.984,A -85,B 0,C 180,E1 -23329.99,E2 -23329.99} C_VEL
LIN {X 0,Y 164.371,Z 234.007,A -85,B 0,C 180,E1 -23336.118,E2 -23336.118} C_VEL
LIN {X 0,Y 164.359,Z 234.01,A -85,B 0,C 180,E1 -23341.218,E2 -23341.218} C_VEL
LIN {X 0,Y 164.281,Z 233.992,A -85,B 0,C 180,E1 -23346.794,E2 -23346.794} C_VEL
LIN {X 0,Y 164.287,Z 233.995,A -85,B 0,C 180,E1 -23349.918,E2 -23349.918} C_VEL
LIN {X 0,Y 164.281,Z 234.013,A -85,B 0,C 180,E1 -23353.342,E2 -23353.342} C_VEL
LIN {X 0,Y 164.263,Z 234.022,A -85,B 0,C 180,E1 -23356.799,E2 -23356.799} C_VEL
LIN {X 0,Y 164.291,Z 234.016,A -85,B 0,C 180,E1 -23360.355,E2 -23360.355} C_VEL
LIN {X 0,Y 164.328,Z 234.007,A -85,B 0,C 180,E1 -23364.352,E2 -23364.352} C_VEL
LIN {X 0,Y 164.373,Z 234.011,A -85,B 0,C 180,E1 -23369.131,E2 -23369.131} C_VEL
LIN {X 0,Y 164.397,Z 233.996,A -85,B 0,C 180,E1 -23374.691,E2 -23374.691} C_VEL
LIN {X 0,Y 164.487,Z 233.994,A -85,B 0,C 180,E1 -23380.052,E2 -23380.052} C_VEL
LIN {X 0,Y 164.5,Z 233.981,A -85,B 0,C 180,E1 -23385.147,E2 -23385.147} C_VEL
LIN {X 0,Y 164.767,Z 233.924,A -85,B 0,C 180,E1 -23390.176,E2 -23390.176} C_VEL
LIN {X 0,Y 164.824,Z 233.928,A -85,B 0,C 180,E1 -23392.651,E2 -23392.651} C_VEL
LIN {X 0,Y 165.041,Z 233.923,A -85,B 0,C 180,E1 -23397.56,E2 -23397.56} C_VEL
LIN {X 0,Y 165.278,Z 233.897,A -85,B 0,C 180,E1 -23400,E2 -23400} C_VEL
LIN {X 0,Y 164.824,Z 233.932,A -85,B 0,C 180,E1 -23407.35,E2 -23407.35} C_VEL
LIN {X 0,Y 164.705,Z 233.961,A -85,B 0,C 180,E1 -23411.059,E2 -23411.059} C_VEL
LIN {X 0,Y 164.443,Z 234.002,A -85,B 0,C 180,E1 -23417.408,E2 -23417.408} C_VEL
LIN {X 0,Y 164.35,Z 234.007,A -85,B 0,C 180,E1 -23422.635,E2 -23422.635} C_VEL
LIN {X 0,Y 164.366,Z 234.014,A -85,B 0,C 180,E1 -23426.112,E2 -23426.112} C_VEL
LIN {X 0,Y 164.36,Z 234.003,A -85,B 0,C 180,E1 -23431.217,E2 -23431.217} C_VEL
LIN {X 0,Y 164.282,Z 234.02,A -85,B 0,C 180,E1 -23436.793,E2 -23436.793} C_VEL
LIN {X 0,Y 164.288,Z 234.023,A -85,B 0,C 180,E1 -23439.918,E2 -23439.918} C_VEL
LIN {X 0,Y 164.326,Z 234.016,A -85,B 0,C 180,E1 -23445.976,E2 -23445.976} C_VEL
LIN {X 0,Y 166.307,Z 242.754,A -85,B 0,C 180,E1 -23450.697,E2 -23450.697} C_VEL
LIN {X 0,Y 173.776,Z 263.829,A -85,B 0,C 180,E1 -23453.103,E2 -23453.103} C_VEL
LIN {X 0,Y 175.988,Z 270.771,A -85,B 0,C 180,E1 -23453.819,E2 -23453.819} C_VEL
LIN {X 0,Y 179.303,Z 312.346,A -85,B 0,C 180,E1 -23456.567,E2 -23456.567} C_VEL
LIN {X 0,Y 176.833,Z 353.91,A -85,B 0,C 180,E1 -23458.64,E2 -23458.64} C_VEL
LIN {X 0,Y 175.677,Z 366.39,A -85,B 0,C 180,E1 -23459.664,E2 -23459.664} C_VEL
LIN {X 0,Y 173.838,Z 379.254,A -85,B 0,C 180,E1 -23461.143,E2 -23461.143} C_VEL
LIN {X 0,Y 171.558,Z 392.281,A -85,B 0,C 180,E1 -23463.216,E2 -23463.216} C_VEL
LIN {X 0,Y 169.401,Z 403.243,A -85,B 0,C 180,E1 -23465.488,E2 -23465.488} C_VEL
LIN {X 0,Y 167.095,Z 414.16,A -85,B 0,C 180,E1 -23468.405,E2 -23468.405} C_VEL
LIN {X 0,Y 165.327,Z 423.08,A -85,B 0,C 180,E1 -23471.408,E2 -23471.408} C_VEL
LIN {X 0,Y 164.241,Z 429.003,A -85,B 0,C 180,E1 -23473.828,E2 -23473.828} C_VEL
LIN {X 0,Y 163.01,Z 432.48,A -85,B 0,C 180,E1 -23475.455,E2 -23475.455} C_VEL
LIN {X 0,Y 159.463,Z 437.397,A -85,B 0,C 180,E1 -23478.25,E2 -23478.25} C_VEL
LIN {X 0,Y 156.255,Z 441.67,A -85,B 0,C 180,E1 -23481.301,E2 -23481.301} C_VEL
LIN {X 0,Y 155.574,Z 444.071,A -85,B 0,C 180,E1 -23483.27,E2 -23483.27} C_VEL
LIN {X 0,Y 155.622,Z 448.287,A -85,B 0,C 180,E1 -23487.411,E2 -23487.411} C_VEL
LIN {X 0,Y 155.942,Z 450.251,A -85,B 0,C 180,E1 -23489.999,E2 -23489.999} C_VEL
LIN {X 0,Y 155.221,Z 452.594,A -85,B 0,C 180,E1 -23495.055,E2 -23495.055} C_VEL
LIN {X 0,Y 155.12,Z 453.228,A -85,B 0,C 180,E1 -23497.811,E2 -23497.811} C_VEL
LIN {X 0,Y 155.846,Z 453.211,A -85,B 0,C 180,E1 -23503.03,E2 -23503.03} C_VEL
LIN {X 0,Y 157.955,Z 451.736,A -85,B 0,C 180,E1 -23508.146,E2 -23508.146} C_VEL
LIN {X 0,Y 159.526,Z 450.445,A -85,B 0,C 180,E1 -23510.636,E2 -23510.636} C_VEL
LIN {X 0,Y 162.489,Z 447.754,A -85,B 0,C 180,E1 -23514.26,E2 -23514.26} C_VEL
LIN {X 0,Y 166.034,Z 444.157,A -85,B 0,C 180,E1 -23517.749,E2 -23517.749} C_VEL
LIN {X 0,Y 170.409,Z 439.561,A -85,B 0,C 180,E1 -23521.032,E2 -23521.032} C_VEL
LIN {X 0,Y 176.426,Z 432.798,A -85,B 0,C 180,E1 -23524.586,E2 -23524.586} C_VEL
LIN {X 0,Y 182.063,Z 425.624,A -85,B 0,C 180,E1 -23527.443,E2 -23527.443} C_VEL
LIN {X 0,Y 188.335,Z 416.821,A -85,B 0,C 180,E1 -23530.068,E2 -23530.068} C_VEL
LIN {X 0,Y 193.954,Z 407.938,A -85,B 0,C 180,E1 -23532.094,E2 -23532.094} C_VEL
LIN {X 0,Y 199.875,Z 397.188,A -85,B 0,C 180,E1 -23533.983,E2 -23533.983} C_VEL
LIN {X 0,Y 205.565,Z 385.134,A -85,B 0,C 180,E1 -23535.535,E2 -23535.535} C_VEL
LIN {X 0,Y 210.14,Z 373.355,A -85,B 0,C 180,E1 -23536.669,E2 -23536.669} C_VEL
LIN {X 0,Y 213.716,Z 361.773,A -85,B 0,C 180,E1 -23537.509,E2 -23537.509} C_VEL
LIN {X 0,Y 216.728,Z 348.254,A -85,B 0,C 180,E1 -23538.23,E2 -23538.23} C_VEL
LIN {X 0,Y 220.05,Z 323.742,A -85,B 0,C 180,E1 -23539.154,E2 -23539.154} C_VEL
LIN {X 0,Y 220.248,Z 319.328,A -85,B 0,C 180,E1 -23539.538,E2 -23539.538} C_VEL
LIN {X 0,Y 218.391,Z 312.789,A -85,B 0,C 180,E1 -23541.713,E2 -23541.713} C_VEL
LIN {X 0,Y 216.907,Z 308.278,A -85,B 0,C 180,E1 -23543.608,E2 -23543.608} C_VEL
LIN {X 0,Y 215.774,Z 304.569,A -85,B 0,C 180,E1 -23545.479,E2 -23545.479} C_VEL
LIN {X 0,Y 214.508,Z 300.746,A -85,B 0,C 180,E1 -23548.006,E2 -23548.006} C_VEL
LIN {X 0,Y 213.38,Z 297.132,A -85,B 0,C 180,E1 -23552.011,E2 -23552.011} C_VEL
LIN {X 0,Y 213.195,Z 296.107,A -85,B 0,C 180,E1 -23554.624,E2 -23554.624} C_VEL
LIN {X 0,Y 213.763,Z 295.977,A -85,B 0,C 180,E1 -23558.044,E2 -23558.044} C_VEL
LIN {X 0,Y 214.446,Z 296.61,A -85,B 0,C 180,E1 -23559.94,E2 -23559.94} C_VEL
LIN {X 0,Y 216.347,Z 299.975,A -85,B 0,C 180,E1 -23563.609,E2 -23563.609} C_VEL
LIN {X 0,Y 218.307,Z 303.745,A -85,B 0,C 180,E1 -23566.267,E2 -23566.267} C_VEL
LIN {X 0,Y 221.393,Z 310.199,A -85,B 0,C 180,E1 -23569.478,E2 -23569.478} C_VEL
LIN {X 0,Y 218.016,Z 336.046,A -85,B 0,C 180,E1 -23570.518,E2 -23570.518} C_VEL
LIN {X 0,Y 215.454,Z 348.757,A -85,B 0,C 180,E1 -23571.335,E2 -23571.335} C_VEL
LIN {X 0,Y 211.869,Z 361.534,A -85,B 0,C 180,E1 -23572.495,E2 -23572.495} C_VEL
LIN {X 0,Y 207.444,Z 373.529,A -85,B 0,C 180,E1 -23573.922,E2 -23573.922} C_VEL
LIN {X 0,Y 202.493,Z 384.346,A -85,B 0,C 180,E1 -23575.589,E2 -23575.589} C_VEL
LIN {X 0,Y 196.218,Z 395.776,A -85,B 0,C 180,E1 -23577.947,E2 -23577.947} C_VEL
LIN {X 0,Y 190.417,Z 404.651,A -85,B 0,C 180,E1 -23580.336,E2 -23580.336} C_VEL
LIN {X 0,Y 184.77,Z 412.134,A -85,B 0,C 180,E1 -23582.999,E2 -23582.999} C_VEL
LIN {X 0,Y 178.851,Z 418.922,A -85,B 0,C 180,E1 -23586.203,E2 -23586.203} C_VEL
LIN {X 0,Y 174.013,Z 423.78,A -85,B 0,C 180,E1 -23589.297,E2 -23589.297} C_VEL
LIN {X 0,Y 168.826,Z 428.189,A -85,B 0,C 180,E1 -23593.236,E2 -23593.236} C_VEL
LIN {X 0,Y 164.459,Z 431.125,A -85,B 0,C 180,E1 -23597.406,E2 -23597.406} C_VEL
LIN {X 0,Y 162.011,Z 432.367,A -85,B 0,C 180,E1 -23600.306,E2 -23600.306} C_VEL
LIN {X 0,Y 159.918,Z 432.986,A -85,B 0,C 180,E1 -23603.299,E2 -23603.299} C_VEL
LIN {X 0,Y 157.858,Z 432.982,A -85,B 0,C 180,E1 -23607.075,E2 -23607.075} C_VEL
LIN {X 0,Y 156.268,Z 431.942,A -85,B 0,C 180,E1 -23611.296,E2 -23611.296} C_VEL
LIN {X 0,Y 155.283,Z 429.518,A -85,B 0,C 180,E1 -23616.041,E2 -23616.041} C_VEL
LIN {X 0,Y 155.171,Z 425.422,A -85,B 0,C 180,E1 -23621.085,E2 -23621.085} C_VEL
LIN {X 0,Y 155.653,Z 421.246,A -85,B 0,C 180,E1 -23624.813,E2 -23624.813} C_VEL
LIN {X 0,Y 156.504,Z 415.977,A -85,B 0,C 180,E1 -23628.511,E2 -23628.511} C_VEL
LIN {X 0,Y 157.844,Z 408.485,A -85,B 0,C 180,E1 -23632.656,E2 -23632.656} C_VEL
LIN {X 0,Y 159.47,Z 400.419,A -85,B 0,C 180,E1 -23636.205,E2 -23636.205} C_VEL
LIN {X 0,Y 161.43,Z 391.459,A -85,B 0,C 180,E1 -23639.371,E2 -23639.371} C_VEL
LIN {X 0,Y 163.74,Z 380.234,A -85,B 0,C 180,E1 -23642.507,E2 -23642.507} C_VEL
LIN {X 0,Y 165.771,Z 369.345,A -85,B 0,C 180,E1 -23644.916,E2 -23644.916} C_VEL
LIN {X 0,Y 167.842,Z 356.483,A -85,B 0,C 180,E1 -23647.102,E2 -23647.102} C_VEL
LIN {X 0,Y 169.551,Z 344.017,A -85,B 0,C 180,E1 -23648.689,E2 -23648.689} C_VEL
LIN {X 0,Y 170.704,Z 330.737,A -85,B 0,C 180,E1 -23649.899,E2 -23649.899} C_VEL
LIN {X 0,Y 171.803,Z 313.047,A -85,B 0,C 180,E1 -23650.898,E2 -23650.898} C_VEL
LIN {X 0,Y 174.172,Z 274.35,A -85,B 0,C 180,E1 -23652.806,E2 -23652.806} C_VEL
LIN {X 0,Y 163.6,Z 248.542,A -85,B 0,C 180,E1 -23655.938,E2 -23655.938} C_VEL
LIN {X 0,Y 157.774,Z 235.816,A -85,B 0,C 180,E1 -23657.775,E2 -23657.775} C_VEL
LIN {X 0,Y 157.594,Z 234.854,A -85,B 0,C 180,E1 -23657.94,E2 -23657.94} C_VEL
LIN {X 0,Y 157.763,Z 234.834,A -85,B 0,C 180,E1 -23662.32,E2 -23662.32} C_VEL
LIN {X 0,Y 158.254,Z 234.771,A -85,B 0,C 180,E1 -23670.001,E2 -23670.001} C_VEL
LIN {X 0,Y 157.763,Z 234.831,A -85,B 0,C 180,E1 -23677.681,E2 -23677.681} C_VEL
LIN {X 0,Y 157.638,Z 234.847,A -85,B 0,C 180,E1 -23681.238,E2 -23681.238} C_VEL
LIN {X 0,Y 157.455,Z 234.871,A -85,B 0,C 180,E1 -23685.535,E2 -23685.535} C_VEL
LIN {X 0,Y 157.368,Z 234.865,A -85,B 0,C 180,E1 -23690.934,E2 -23690.934} C_VEL
LIN {X 0,Y 157.311,Z 234.887,A -85,B 0,C 180,E1 -23696.681,E2 -23696.681} C_VEL
LIN {X 0,Y 157.269,Z 234.888,A -85,B 0,C 180,E1 -23702.43,E2 -23702.43} C_VEL
LIN {X 0,Y 157.259,Z 234.867,A -85,B 0,C 180,E1 -23706.445,E2 -23706.445} C_VEL
LIN {X 0,Y 157.192,Z 234.892,A -85,B 0,C 180,E1 -23712.118,E2 -23712.118} C_VEL
LIN {X 0,Y 157.192,Z 234.904,A -85,B 0,C 180,E1 -23717.883,E2 -23717.883} C_VEL
LIN {X 0,Y 157.261,Z 234.886,A -85,B 0,C 180,E1 -23723.556,E2 -23723.556} C_VEL
LIN {X 0,Y 157.285,Z 234.892,A -85,B 0,C 180,E1 -23728.103,E2 -23728.103} C_VEL
LIN {X 0,Y 157.311,Z 234.879,A -85,B 0,C 180,E1 -23733.464,E2 -23733.464} C_VEL
LIN {X 0,Y 157.394,Z 234.877,A -85,B 0,C 180,E1 -23739.671,E2 -23739.671} C_VEL
LIN {X 0,Y 157.438,Z 234.864,A -85,B 0,C 180,E1 -23744.464,E2 -23744.464} C_VEL
LIN {X 0,Y 157.689,Z 234.805,A -85,B 0,C 180,E1 -23749.731,E2 -23749.731} C_VEL
LIN {X 0,Y 157.762,Z 234.804,A -85,B 0,C 180,E1 -23752.32,E2 -23752.32} C_VEL
LIN {X 0,Y 158.24,Z 234.774,A -85,B 0,C 180,E1 -23760,E2 -23760} C_VEL
LIN {X 0,Y 157.762,Z 234.809,A -85,B 0,C 180,E1 -23767.68,E2 -23767.68} C_VEL
LIN {X 0,Y 157.635,Z 234.841,A -85,B 0,C 180,E1 -23771.227,E2 -23771.227} C_VEL
LIN {X 0,Y 157.42,Z 234.878,A -85,B 0,C 180,E1 -23775.538,E2 -23775.538} C_VEL
LIN {X 0,Y 157.311,Z 234.876,A -85,B 0,C 180,E1 -23780.941,E2 -23780.941} C_VEL
LIN {X 0,Y 157.294,Z 234.894,A -85,B 0,C 180,E1 -23786.668,E2 -23786.668} C_VEL
LIN {X 0,Y 157.27,Z 234.893,A -85,B 0,C 180,E1 -23792.429,E2 -23792.429} C_VEL
LIN {X 0,Y 157.261,Z 234.895,A -85,B 0,C 180,E1 -23796.444,E2 -23796.444} C_VEL
LIN {X 0,Y 157.192,Z 234.908,A -85,B 0,C 180,E1 -23802.117,E2 -23802.117} C_VEL
LIN {X 0,Y 157.265,Z 235.063,A -85,B 0,C 180,E1 -23805.452,E2 -23805.452} C_VEL
LIN {X 0,Y 159.015,Z 242.475,A -85,B 0,C 180,E1 -23809.433,E2 -23809.433} C_VEL
LIN {X 0,Y 166.151,Z 262.197,A -85,B 0,C 180,E1 -23811.859,E2 -23811.859} C_VEL
LIN {X 0,Y 169.477,Z 272.266,A -85,B 0,C 180,E1 -23812.966,E2 -23812.966} C_VEL
LIN {X 0,Y 172.625,Z 312.96,A -85,B 0,C 180,E1 -23815.775,E2 -23815.775} C_VEL
LIN {X 0,Y 170.15,Z 353.411,A -85,B 0,C 180,E1 -23817.872,E2 -23817.872} C_VEL
LIN {X 0,Y 168.851,Z 366.557,A -85,B 0,C 180,E1 -23818.996,E2 -23818.996} C_VEL
LIN {X 0,Y 167.124,Z 378.218,A -85,B 0,C 180,E1 -23820.388,E2 -23820.388} C_VEL
LIN {X 0,Y 164.911,Z 390.579,A -85,B 0,C 180,E1 -23822.389,E2 -23822.389} C_VEL
LIN {X 0,Y 162.69,Z 401.696,A -85,B 0,C 180,E1 -23824.737,E2 -23824.737} C_VEL
LIN {X 0,Y 160.506,Z 411.874,A -85,B 0,C 180,E1 -23827.471,E2 -23827.471} C_VEL
LIN {X 0,Y 158.528,Z 421.031,A -85,B 0,C 180,E1 -23830.579,E2 -23830.579} C_VEL
LIN {X 0,Y 156.965,Z 430.016,A -85,B 0,C 180,E1 -23834.416,E2 -23834.416} C_VEL
LIN {X 0,Y 155.901,Z 437.126,A -85,B 0,C 180,E1 -23838.295,E2 -23838.295} C_VEL
LIN {X 0,Y 155.57,Z 442.768,A -85,B 0,C 180,E1 -23842.21,E2 -23842.21} C_VEL
LIN {X 0,Y 155.574,Z 444.071,A -85,B 0,C 180,E1 -23843.27,E2 -23843.27} C_VEL
LIN {X 0,Y 154.933,Z 446.247,A -85,B 0,C 180,E1 -23845.28,E2 -23845.28} C_VEL
LIN {X 0,Y 153.336,Z 447.931,A -85,B 0,C 180,E1 -23847.32,E2 -23847.32} C_VEL
LIN {X 0,Y 149.482,Z 450.321,A -85,B 0,C 180,E1 -23851.579,E2 -23851.579} C_VEL
LIN {X 0,Y 148.19,Z 451.514,A -85,B 0,C 180,E1 -23854.617,E2 -23854.617} C_VEL
LIN {X 0,Y 148.089,Z 452.485,A -85,B 0,C 180,E1 -23858.184,E2 -23858.184} C_VEL
LIN {X 0,Y 148.903,Z 452.708,A -85,B 0,C 180,E1 -23863.649,E2 -23863.649} C_VEL
LIN {X 0,Y 151.194,Z 451.409,A -85,B 0,C 180,E1 -23868.988,E2 -23868.988} C_VEL
LIN {X 0,Y 154.92,Z 448.662,A -85,B 0,C 180,E1 -23874.097,E2 -23874.097} C_VEL
LIN {X 0,Y 158.405,Z 445.552,A -85,B 0,C 180,E1 -23877.765,E2 -23877.765} C_VEL
LIN {X 0,Y 162.751,Z 441.502,A -85,B 0,C 180,E1 -23881.21,E2 -23881.21} C_VEL
LIN {X 0,Y 167.878,Z 436.443,A -85,B 0,C 180,E1 -23884.413,E2 -23884.413} C_VEL
LIN {X 0,Y 174.561,Z 429.066,A -85,B 0,C 180,E1 -23887.877,E2 -23887.877} C_VEL
LIN {X 0,Y 180.821,Z 421.18,A -85,B 0,C 180,E1 -23890.618,E2 -23890.618} C_VEL
LIN {X 0,Y 187.655,Z 411.553,A -85,B 0,C 180,E1 -23893.116,E2 -23893.116} C_VEL
LIN {X 0,Y 194.307,Z 400.749,A -85,B 0,C 180,E1 -23895.22,E2 -23895.22} C_VEL
LIN {X 0,Y 200.102,Z 389.721,A -85,B 0,C 180,E1 -23896.784,E2 -23896.784} C_VEL
LIN {X 0,Y 205.459,Z 377.513,A -85,B 0,C 180,E1 -23898.071,E2 -23898.071} C_VEL
LIN {X 0,Y 209.859,Z 364.707,A -85,B 0,C 180,E1 -23899.077,E2 -23899.077} C_VEL
LIN {X 0,Y 213.465,Z 350.68,A -85,B 0,C 180,E1 -23899.872,E2 -23899.872} C_VEL
LIN {X 0,Y 215.975,Z 335.31,A -85,B 0,C 180,E1 -23900.472,E2 -23900.472} C_VEL
LIN {X 0,Y 217.46,Z 323.55,A -85,B 0,C 180,E1 -23900.945,E2 -23900.945} C_VEL
LIN {X 0,Y 216.096,Z 318.231,A -85,B 0,C 180,E1 -23902.775,E2 -23902.775} C_VEL
LIN {X 0,Y 214.981,Z 314.275,A -85,B 0,C 180,E1 -23904.477,E2 -23904.477} C_VEL
LIN {X 0,Y 214.107,Z 311.08,A -85,B 0,C 180,E1 -23906.081,E2 -23906.081} C_VEL
LIN {X 0,Y 213.026,Z 307.36,A -85,B 0,C 180,E1 -23908.574,E2 -23908.574} C_VEL
LIN {X 0,Y 212.115,Z 304.018,A -85,B 0,C 180,E1 -23912.363,E2 -23912.363} C_VEL
LIN {X 0,Y 212.08,Z 302.966,A -85,B 0,C 180,E1 -23915.661,E2 -23915.661} C_VEL
LIN {X 0,Y 212.91,Z 303.17,A -85,B 0,C 180,E1 -23919.124,E2 -23919.124} C_VEL
LIN {X 0,Y 214.724,Z 306.611,A -85,B 0,C 180,E1 -23923.082,E2 -23923.082} C_VEL
LIN {X 0,Y 216.512,Z 310.331,A -85,B 0,C 180,E1 -23925.704,E2 -23925.704} C_VEL
LIN {X 0,Y 218.386,Z 314.673,A -85,B 0,C 180,E1 -23927.892,E2 -23927.892} C_VEL
LIN {X 0,Y 215.153,Z 337.667,A -85,B 0,C 180,E1 -23928.836,E2 -23928.836} C_VEL
LIN {X 0,Y 212.314,Z 350.666,A -85,B 0,C 180,E1 -23929.697,E2 -23929.697} C_VEL
LIN {X 0,Y 208.254,Z 363.777,A -85,B 0,C 180,E1 -23930.903,E2 -23930.903} C_VEL
LIN {X 0,Y 203.726,Z 375.379,A -85,B 0,C 180,E1 -23932.318,E2 -23932.318} C_VEL
LIN {X 0,Y 198.736,Z 385.623,A -85,B 0,C 180,E1 -23933.91,E2 -23933.91} C_VEL
LIN {X 0,Y 193.279,Z 395.119,A -85,B 0,C 180,E1 -23935.829,E2 -23935.829} C_VEL
LIN {X 0,Y 187.987,Z 403.022,A -85,B 0,C 180,E1 -23937.857,E2 -23937.857} C_VEL
LIN {X 0,Y 181.717,Z 411.174,A -85,B 0,C 180,E1 -23940.553,E2 -23940.553} C_VEL
LIN {X 0,Y 175.072,Z 418.559,A -85,B 0,C 180,E1 -23943.866,E2 -23943.866} C_VEL
LIN {X 0,Y 169.489,Z 423.87,A -85,B 0,C 180,E1 -23947.146,E2 -23947.146} C_VEL
LIN {X 0,Y 164.467,Z 427.93,A -85,B 0,C 180,E1 -23950.634,E2 -23950.634} C_VEL
LIN {X 0,Y 159.789,Z 431.064,A -85,B 0,C 180,E1 -23954.622,E2 -23954.622} C_VEL
LIN {X 0,Y 155.894,Z 432.964,A -85,B 0,C 180,E1 -23958.789,E2 -23958.789} C_VEL
LIN {X 0,Y 152.798,Z 433.699,A -85,B 0,C 180,E1 -23963.089,E2 -23963.089} C_VEL
LIN {X 0,Y 150.332,Z 433.233,A -85,B 0,C 180,E1 -23967.872,E2 -23967.872} C_VEL
LIN {X 0,Y 148.969,Z 431.905,A -85,B 0,C 180,E1 -23971.877,E2 -23971.877} C_VEL
LIN {X 0,Y 148.164,Z 429.44,A -85,B 0,C 180,E1 -23976.258,E2 -23976.258} C_VEL
LIN {X 0,Y 148.047,Z 425.94,A -85,B 0,C 180,E1 -23980.577,E2 -23980.577} C_VEL
LIN {X 0,Y 148.603,Z 420.881,A -85,B 0,C 180,E1 -23985.187,E2 -23985.187} C_VEL
LIN {X 0,Y 149.718,Z 414.391,A -85,B 0,C 180,E1 -23989.71,E2 -23989.71} C_VEL
LIN {X 0,Y 151.254,Z 406.466,A -85,B 0,C 180,E1 -23993.983,E2 -23993.983} C_VEL
LIN {X 0,Y 153.103,Z 397.826,A -85,B 0,C 180,E1 -23997.656,E2 -23997.656} C_VEL
LIN {X 0,Y 155.132,Z 388.461,A -85,B 0,C 180,E1 -24000.856,E2 -24000.856} C_VEL
LIN {X 0,Y 157.478,Z 377.29,A -85,B 0,C 180,E1 -24003.863,E2 -24003.863} C_VEL
LIN {X 0,Y 159.585,Z 365.765,A -85,B 0,C 180,E1 -24006.306,E2 -24006.306} C_VEL
LIN {X 0,Y 161.606,Z 353.41,A -85,B 0,C 180,E1 -24008.306,E2 -24008.306} C_VEL
LIN {X 0,Y 163.343,Z 339.391,A -85,B 0,C 180,E1 -24009.97,E2 -24009.97} C_VEL
LIN {X 0,Y 164.401,Z 325.888,A -85,B 0,C 180,E1 -24011.052,E2 -24011.052} C_VEL
LIN {X 0,Y 167.511,Z 275.953,A -85,B 0,C 180,E1 -24013.644,E2 -24013.644} C_VEL
LIN {X 0,Y 157.558,Z 251.549,A -85,B 0,C 180,E1 -24016.786,E2 -24016.786} C_VEL
LIN {X 0,Y 150.784,Z 236.515,A -85,B 0,C 180,E1 -24019.045,E2 -24019.045} C_VEL
LIN {X 0,Y 150.635,Z 235.723,A -85,B 0,C 180,E1 -24019.14,E2 -24019.14} C_VEL
LIN {X 0,Y 150.702,Z 235.714,A -85,B 0,C 180,E1 -24021.958,E2 -24021.958} C_VEL
LIN {X 0,Y 151.214,Z 235.648,A -85,B 0,C 180,E1 -24030.001,E2 -24030.001} C_VEL
LIN {X 0,Y 150.702,Z 235.712,A -85,B 0,C 180,E1 -24038.043,E2 -24038.043} C_VEL
LIN {X 0,Y 150.578,Z 235.727,A -85,B 0,C 180,E1 -24041.438,E2 -24041.438} C_VEL
LIN {X 0,Y 150.363,Z 235.755,A -85,B 0,C 180,E1 -24046.287,E2 -24046.287} C_VEL
LIN {X 0,Y 150.351,Z 235.739,A -85,B 0,C 180,E1 -24050.791,E2 -24050.791} C_VEL
LIN {X 0,Y 150.24,Z 235.769,A -85,B 0,C 180,E1 -24057.278,E2 -24057.278} C_VEL
LIN {X 0,Y 150.209,Z 235.767,A -85,B 0,C 180,E1 -24062.629,E2 -24062.629} C_VEL
LIN {X 0,Y 150.17,Z 235.743,A -85,B 0,C 180,E1 -24067.475,E2 -24067.475} C_VEL
LIN {X 0,Y 150.134,Z 235.765,A -85,B 0,C 180,E1 -24071.498,E2 -24071.498} C_VEL
LIN {X 0,Y 150.128,Z 235.782,A -85,B 0,C 180,E1 -24075.396,E2 -24075.396} C_VEL
LIN {X 0,Y 150.139,Z 235.783,A -85,B 0,C 180,E1 -24079.055,E2 -24079.055} C_VEL
LIN {X 0,Y 150.177,Z 235.768,A -85,B 0,C 180,E1 -24082.71,E2 -24082.71} C_VEL
LIN {X 0,Y 150.21,Z 235.774,A -85,B 0,C 180,E1 -24087.373,E2 -24087.373} C_VEL
LIN {X 0,Y 150.241,Z 235.763,A -85,B 0,C 180,E1 -24092.723,E2 -24092.723} C_VEL
LIN {X 0,Y 150.351,Z 235.755,A -85,B 0,C 180,E1 -24099.211,E2 -24099.211} C_VEL
LIN {X 0,Y 150.35,Z 235.749,A -85,B 0,C 180,E1 -24103.712,E2 -24103.712} C_VEL
LIN {X 0,Y 150.61,Z 235.687,A -85,B 0,C 180,E1 -24109.243,E2 -24109.243} C_VEL
LIN {X 0,Y 150.685,Z 235.683,A -85,B 0,C 180,E1 -24111.957,E2 -24111.957} C_VEL
LIN {X 0,Y 151.201,Z 235.651,A -85,B 0,C 180,E1 -24120,E2 -24120} C_VEL
LIN {X 0,Y 150.685,Z 235.69,A -85,B 0,C 180,E1 -24128.043,E2 -24128.043} C_VEL
LIN {X 0,Y 150.577,Z 235.721,A -85,B 0,C 180,E1 -24131.431,E2 -24131.431} C_VEL
LIN {X 0,Y 150.325,Z 235.761,A -85,B 0,C 180,E1 -24136.291,E2 -24136.291} C_VEL
LIN {X 0,Y 150.286,Z 235.751,A -85,B 0,C 180,E1 -24140.724,E2 -24140.724} C_VEL
LIN {X 0,Y 150.23,Z 235.775,A -85,B 0,C 180,E1 -24147.269,E2 -24147.269} C_VEL
LIN {X 0,Y 150.21,Z 235.772,A -85,B 0,C 180,E1 -24152.628,E2 -24152.628} C_VEL
LIN {X 0,Y 150.171,Z 235.781,A -85,B 0,C 180,E1 -24157.474,E2 -24157.474} C_VEL
LIN {X 0,Y 150.155,Z 235.785,A -85,B 0,C 180,E1 -24163.746,E2 -24163.746} C_VEL
LIN {X 0,Y 150.193,Z 235.782,A -85,B 0,C 180,E1 -24164.58,E2 -24164.58} C_VEL
LIN {X 0,Y 151.564,Z 241.67,A -85,B 0,C 180,E1 -24167.996,E2 -24167.996} C_VEL
LIN {X 0,Y 159.24,Z 262.558,A -85,B 0,C 180,E1 -24170.774,E2 -24170.774} C_VEL
LIN {X 0,Y 163.108,Z 274.611,A -85,B 0,C 180,E1 -24172.16,E2 -24172.16} C_VEL
LIN {X 0,Y 165.943,Z 313.896,A -85,B 0,C 180,E1 -24174.963,E2 -24174.963} C_VEL
LIN {X 0,Y 163.491,Z 352.411,A -85,B 0,C 180,E1 -24177.039,E2 -24177.039} C_VEL
LIN {X 0,Y 162.263,Z 364.979,A -85,B 0,C 180,E1 -24178.137,E2 -24178.137} C_VEL
LIN {X 0,Y 160.295,Z 377.892,A -85,B 0,C 180,E1 -24179.72,E2 -24179.72} C_VEL
LIN {X 0,Y 158.032,Z 390.177,A -85,B 0,C 180,E1 -24181.802,E2 -24181.802} C_VEL
LIN {X 0,Y 155.762,Z 401.201,A -85,B 0,C 180,E1 -24184.229,E2 -24184.229} C_VEL
LIN {X 0,Y 153.502,Z 411.423,A -85,B 0,C 180,E1 -24187.096,E2 -24187.096} C_VEL
LIN {X 0,Y 151.494,Z 420.573,A -85,B 0,C 180,E1 -24190.345,E2 -24190.345} C_VEL
LIN {X 0,Y 149.9,Z 429.546,A -85,B 0,C 180,E1 -24194.36,E2 -24194.36} C_VEL
LIN {X 0,Y 148.829,Z 436.636,A -85,B 0,C 180,E1 -24198.422,E2 -24198.422} C_VEL
LIN {X 0,Y 148.515,Z 441.44,A -85,B 0,C 180,E1 -24201.838,E2 -24201.838} C_VEL
LIN {X 0,Y 148.578,Z 445.969,A -85,B 0,C 180,E1 -24205.931,E2 -24205.931} C_VEL
LIN {X 0,Y 148.886,Z 449.286,A -85,B 0,C 180,E1 -24209.999,E2 -24209.999} C_VEL
LIN {X 0,Y 148.19,Z 451.514,A -85,B 0,C 180,E1 -24214.617,E2 -24214.617} C_VEL
LIN {X 0,Y 147.441,Z 452.183,A -85,B 0,C 180,E1 -24216.869,E2 -24216.869} C_VEL
LIN {X 0,Y 144.8,Z 452.464,A -85,B 0,C 180,E1 -24220.614,E2 -24220.614} C_VEL
LIN {X 0,Y 142.959,Z 452.25,A -85,B 0,C 180,E1 -24223.708,E2 -24223.708} C_VEL
LIN {X 0,Y 142.647,Z 451.961,A -85,B 0,C 180,E1 -24226.086,E2 -24226.086} C_VEL
LIN {X 0,Y 142.865,Z 451.831,A -85,B 0,C 180,E1 -24226.875,E2 -24226.875} C_VEL
LIN {X 0,Y 144.474,Z 451.094,A -85,B 0,C 180,E1 -24229.908,E2 -24229.908} C_VEL
LIN {X 0,Y 148.43,Z 448.532,A -85,B 0,C 180,E1 -24235.222,E2 -24235.222} C_VEL
LIN {X 0,Y 152.147,Z 445.638,A -85,B 0,C 180,E1 -24239.013,E2 -24239.013} C_VEL
LIN {X 0,Y 156.732,Z 441.834,A -85,B 0,C 180,E1 -24242.553,E2 -24242.553} C_VEL
LIN {X 0,Y 162.087,Z 437.003,A -85,B 0,C 180,E1 -24245.827,E2 -24245.827} C_VEL
LIN {X 0,Y 169.065,Z 429.889,A -85,B 0,C 180,E1 -24249.34,E2 -24249.34} C_VEL
LIN {X 0,Y 175.564,Z 422.421,A -85,B 0,C 180,E1 -24252.106,E2 -24252.106} C_VEL
LIN {X 0,Y 182.626,Z 413.291,A -85,B 0,C 180,E1 -24254.612,E2 -24254.612} C_VEL
LIN {X 0,Y 189.472,Z 402.948,A -85,B 0,C 180,E1 -24256.713,E2 -24256.713} C_VEL
LIN {X 0,Y 196.099,Z 391.366,A -85,B 0,C 180,E1 -24258.429,E2 -24258.429} C_VEL
LIN {X 0,Y 201.606,Z 379.793,A -85,B 0,C 180,E1 -24259.69,E2 -24259.69} C_VEL
LIN {X 0,Y 206.467,Z 366.991,A -85,B 0,C 180,E1 -24260.749,E2 -24260.749} C_VEL
LIN {X 0,Y 210.254,Z 353.872,A -85,B 0,C 180,E1 -24261.527,E2 -24261.527} C_VEL
LIN {X 0,Y 213.135,Z 338.982,A -85,B 0,C 180,E1 -24262.144,E2 -24262.144} C_VEL
LIN {X 0,Y 214.743,Z 327.06,A -85,B 0,C 180,E1 -24262.583,E2 -24262.583} C_VEL
LIN {X 0,Y 213.4,Z 321.402,A -85,B 0,C 180,E1 -24264.819,E2 -24264.819} C_VEL
LIN {X 0,Y 212.327,Z 317.213,A -85,B 0,C 180,E1 -24266.952,E2 -24266.952} C_VEL
LIN {X 0,Y 211.536,Z 313.922,A -85,B 0,C 180,E1 -24269.222,E2 -24269.222} C_VEL
LIN {X 0,Y 210.851,Z 310.886,A -85,B 0,C 180,E1 -24272.773,E2 -24272.773} C_VEL
LIN {X 0,Y 210.851,Z 309.978,A -85,B 0,C 180,E1 -24275.51,E2 -24275.51} C_VEL
LIN {X 0,Y 211.704,Z 310.286,A -85,B 0,C 180,E1 -24279.192,E2 -24279.192} C_VEL
LIN {X 0,Y 213.159,Z 313.364,A -85,B 0,C 180,E1 -24282.626,E2 -24282.626} C_VEL
LIN {X 0,Y 214.809,Z 316.964,A -85,B 0,C 180,E1 -24285.181,E2 -24285.181} C_VEL
LIN {X 0,Y 215.578,Z 319.012,A -85,B 0,C 180,E1 -24286.275,E2 -24286.275} C_VEL
LIN {X 0,Y 212.637,Z 338.819,A -85,B 0,C 180,E1 -24287.089,E2 -24287.089} C_VEL
LIN {X 0,Y 209.628,Z 351.845,A -85,B 0,C 180,E1 -24287.944,E2 -24287.944} C_VEL
LIN {X 0,Y 205.357,Z 365.032,A -85,B 0,C 180,E1 -24289.149,E2 -24289.149} C_VEL
LIN {X 0,Y 200.466,Z 376.725,A -85,B 0,C 180,E1 -24290.573,E2 -24290.573} C_VEL
LIN {X 0,Y 194.983,Z 387.255,A -85,B 0,C 180,E1 -24292.227,E2 -24292.227} C_VEL
LIN {X 0,Y 188.576,Z 397.696,A -85,B 0,C 180,E1 -24294.386,E2 -24294.386} C_VEL
LIN {X 0,Y 181.728,Z 406.954,A -85,B 0,C 180,E1 -24296.926,E2 -24296.926} C_VEL
LIN {X 0,Y 174.607,Z 415.176,A -85,B 0,C 180,E1 -24300,E2 -24300} C_VEL
LIN {X 0,Y 168.878,Z 420.805,A -85,B 0,C 180,E1 -24302.841,E2 -24302.841} C_VEL
LIN {X 0,Y 162.681,Z 426.064,A -85,B 0,C 180,E1 -24306.477,E2 -24306.477} C_VEL
LIN {X 0,Y 157.172,Z 429.922,A -85,B 0,C 180,E1 -24310.351,E2 -24310.351} C_VEL
LIN {X 0,Y 152.427,Z 432.52,A -85,B 0,C 180,E1 -24314.478,E2 -24314.478} C_VEL
LIN {X 0,Y 148.056,Z 434.078,A -85,B 0,C 180,E1 -24319.407,E2 -24319.407} C_VEL
LIN {X 0,Y 145.419,Z 434.27,A -85,B 0,C 180,E1 -24323.329,E2 -24323.329} C_VEL
LIN {X 0,Y 143.149,Z 433.501,A -85,B 0,C 180,E1 -24327.907,E2 -24327.907} C_VEL
LIN {X 0,Y 141.546,Z 431.387,A -85,B 0,C 180,E1 -24333.105,E2 -24333.105} C_VEL
LIN {X 0,Y 140.912,Z 427.62,A -85,B 0,C 180,E1 -24338.656,E2 -24338.656} C_VEL
LIN {X 0,Y 141.144,Z 423.747,A -85,B 0,C 180,E1 -24342.769,E2 -24342.769} C_VEL
LIN {X 0,Y 142.105,Z 417.441,A -85,B 0,C 180,E1 -24347.889,E2 -24347.889} C_VEL
LIN {X 0,Y 143.42,Z 410.239,A -85,B 0,C 180,E1 -24352.352,E2 -24352.352} C_VEL
LIN {X 0,Y 145.002,Z 402.618,A -85,B 0,C 180,E1 -24356.126,E2 -24356.126} C_VEL
LIN {X 0,Y 147.245,Z 393.006,A -85,B 0,C 180,E1 -24359.932,E2 -24359.932} C_VEL
LIN {X 0,Y 149.544,Z 382.349,A -85,B 0,C 180,E1 -24363.243,E2 -24363.243} C_VEL
LIN {X 0,Y 151.852,Z 371.137,A -85,B 0,C 180,E1 -24365.987,E2 -24365.987} C_VEL
LIN {X 0,Y 153.999,Z 358.985,A -85,B 0,C 180,E1 -24368.289,E2 -24368.289} C_VEL
LIN {X 0,Y 155.993,Z 345.631,A -85,B 0,C 180,E1 -24370.16,E2 -24370.16} C_VEL
LIN {X 0,Y 157.263,Z 332.468,A -85,B 0,C 180,E1 -24371.482,E2 -24371.482} C_VEL
LIN {X 0,Y 158.579,Z 313.064,A -85,B 0,C 180,E1 -24372.666,E2 -24372.666} C_VEL
LIN {X 0,Y 160.989,Z 277.851,A -85,B 0,C 180,E1 -24374.521,E2 -24374.521} C_VEL
LIN {X 0,Y 152.017,Z 255.551,A -85,B 0,C 180,E1 -24377.497,E2 -24377.497} C_VEL
LIN {X 0,Y 143.777,Z 237.519,A -85,B 0,C 180,E1 -24380.416,E2 -24380.416} C_VEL
LIN {X 0,Y 143.579,Z 236.602,A -85,B 0,C 180,E1 -24380.581,E2 -24380.581} C_VEL
LIN {X 0,Y 143.816,Z 236.569,A -85,B 0,C 180,E1 -24387.2,E2 -24387.2} C_VEL
LIN {X 0,Y 144.173,Z 236.525,A -85,B 0,C 180,E1 -24390.001,E2 -24390.001} C_VEL
LIN {X 0,Y 143.624,Z 236.594,A -85,B 0,C 180,E1 -24398.442,E2 -24398.442} C_VEL
LIN {X 0,Y 143.507,Z 236.608,A -85,B 0,C 180,E1 -24401.631,E2 -24401.631} C_VEL
LIN {X 0,Y 143.303,Z 236.633,A -85,B 0,C 180,E1 -24407.114,E2 -24407.114} C_VEL
LIN {X 0,Y 143.276,Z 236.617,A -85,B 0,C 180,E1 -24411.253,E2 -24411.253} C_VEL
LIN {X 0,Y 143.184,Z 236.65,A -85,B 0,C 180,E1 -24417.932,E2 -24417.932} C_VEL
LIN {X 0,Y 143.139,Z 236.642,A -85,B 0,C 180,E1 -24423.417,E2 -24423.417} C_VEL
LIN {X 0,Y 143.053,Z 236.634,A -85,B 0,C 180,E1 -24429.694,E2 -24429.694} C_VEL
LIN {X 0,Y 143.035,Z 236.658,A -85,B 0,C 180,E1 -24433.464,E2 -24433.464} C_VEL
LIN {X 0,Y 143.039,Z 236.668,A -85,B 0,C 180,E1 -24437.478,E2 -24437.478} C_VEL
LIN {X 0,Y 143.073,Z 236.654,A -85,B 0,C 180,E1 -24441.81,E2 -24441.81} C_VEL
LIN {X 0,Y 143.178,Z 236.65,A -85,B 0,C 180,E1 -24447.32,E2 -24447.32} C_VEL
LIN {X 0,Y 143.185,Z 236.644,A -85,B 0,C 180,E1 -24452.07,E2 -24452.07} C_VEL
LIN {X 0,Y 143.277,Z 236.636,A -85,B 0,C 180,E1 -24458.749,E2 -24458.749} C_VEL
LIN {X 0,Y 143.294,Z 236.63,A -85,B 0,C 180,E1 -24462.886,E2 -24462.886} C_VEL
LIN {X 0,Y 143.536,Z 236.569,A -85,B 0,C 180,E1 -24468.706,E2 -24468.706} C_VEL
LIN {X 0,Y 143.61,Z 236.559,A -85,B 0,C 180,E1 -24471.558,E2 -24471.558} C_VEL
LIN {X 0,Y 144.159,Z 236.528,A -85,B 0,C 180,E1 -24480,E2 -24480} C_VEL
LIN {X 0,Y 143.611,Z 236.57,A -85,B 0,C 180,E1 -24488.443,E2 -24488.443} C_VEL
LIN {X 0,Y 143.503,Z 236.602,A -85,B 0,C 180,E1 -24491.619,E2 -24491.619} C_VEL
LIN {X 0,Y 143.262,Z 236.64,A -85,B 0,C 180,E1 -24497.118,E2 -24497.118} C_VEL
LIN {X 0,Y 143.224,Z 236.629,A -85,B 0,C 180,E1 -24501.197,E2 -24501.197} C_VEL
LIN {X 0,Y 143.178,Z 236.651,A -85,B 0,C 180,E1 -24507.926,E2 -24507.926} C_VEL
LIN {X 0,Y 143.14,Z 236.654,A -85,B 0,C 180,E1 -24513.416,E2 -24513.416} C_VEL
LIN {X 0,Y 143.054,Z 236.668,A -85,B 0,C 180,E1 -24519.693,E2 -24519.693} C_VEL
LIN {X 0,Y 143.122,Z 236.742,A -85,B 0,C 180,E1 -24523.795,E2 -24523.795} C_VEL
LIN {X 0,Y 144.236,Z 241.356,A -85,B 0,C 180,E1 -24526.507,E2 -24526.507} C_VEL
LIN {X 0,Y 151.213,Z 259.705,A -85,B 0,C 180,E1 -24529.168,E2 -24529.168} C_VEL
LIN {X 0,Y 156.641,Z 276.053,A -85,B 0,C 180,E1 -24531.215,E2 -24531.215} C_VEL
LIN {X 0,Y 159.341,Z 313.43,A -85,B 0,C 180,E1 -24534.033,E2 -24534.033} C_VEL
LIN {X 0,Y 156.793,Z 352.203,A -85,B 0,C 180,E1 -24536.213,E2 -24536.213} C_VEL
LIN {X 0,Y 155.34,Z 366.061,A -85,B 0,C 180,E1 -24537.502,E2 -24537.502} C_VEL
LIN {X 0,Y 153.501,Z 377.522,A -85,B 0,C 180,E1 -24538.997,E2 -24538.997} C_VEL
LIN {X 0,Y 151.176,Z 389.774,A -85,B 0,C 180,E1 -24541.162,E2 -24541.162} C_VEL
LIN {X 0,Y 148.776,Z 401.011,A -85,B 0,C 180,E1 -24543.751,E2 -24543.751} C_VEL
LIN {X 0,Y 146.521,Z 410.978,A -85,B 0,C 180,E1 -24546.688,E2 -24546.688} C_VEL
LIN {X 0,Y 144.454,Z 420.112,A -85,B 0,C 180,E1 -24550.088,E2 -24550.088} C_VEL
LIN {X 0,Y 142.816,Z 429.07,A -85,B 0,C 180,E1 -24554.296,E2 -24554.296} C_VEL
LIN {X 0,Y 141.758,Z 436.132,A -85,B 0,C 180,E1 -24558.561,E2 -24558.561} C_VEL
LIN {X 0,Y 141.508,Z 442.299,A -85,B 0,C 180,E1 -24563.368,E2 -24563.368} C_VEL
LIN {X 0,Y 141.564,Z 446.008,A -85,B 0,C 180,E1 -24567.154,E2 -24567.154} C_VEL
LIN {X 0,Y 141.831,Z 448.208,A -85,B 0,C 180,E1 -24569.999,E2 -24569.999} C_VEL
LIN {X 0,Y 141.125,Z 450.774,A -85,B 0,C 180,E1 -24575.123,E2 -24575.123} C_VEL
LIN {X 0,Y 141.059,Z 451.734,A -85,B 0,C 180,E1 -24578.595,E2 -24578.595} C_VEL
LIN {X 0,Y 141.988,Z 452.137,A -85,B 0,C 180,E1 -24584.328,E2 -24584.328} C_VEL
LIN {X 0,Y 142.865,Z 451.831,A -85,B 0,C 180,E1 -24586.875,E2 -24586.875} C_VEL
LIN {X 0,Y 143.296,Z 451.398,A -85,B 0,C 180,E1 -24589.232,E2 -24589.232} C_VEL
LIN {X 0,Y 142.862,Z 450.084,A -85,B 0,C 180,E1 -24593.17,E2 -24593.17} C_VEL
LIN {X 0,Y 143.166,Z 448.089,A -85,B 0,C 180,E1 -24597.057,E2 -24597.057} C_VEL
LIN {X 0,Y 144.708,Z 446.591,A -85,B 0,C 180,E1 -24599.246,E2 -24599.246} C_VEL
LIN {X 0,Y 150.815,Z 442.093,A -85,B 0,C 180,E1 -24604,E2 -24604} C_VEL
LIN {X 0,Y 156.411,Z 437.504,A -85,B 0,C 180,E1 -24607.343,E2 -24607.343} C_VEL
LIN {X 0,Y 163.688,Z 430.805,A -85,B 0,C 180,E1 -24610.901,E2 -24610.901} C_VEL
LIN {X 0,Y 170.434,Z 423.642,A -85,B 0,C 180,E1 -24613.685,E2 -24613.685} C_VEL
LIN {X 0,Y 177.724,Z 414.874,A -85,B 0,C 180,E1 -24616.193,E2 -24616.193} C_VEL
LIN {X 0,Y 185.451,Z 404.215,A -85,B 0,C 180,E1 -24618.457,E2 -24618.457} C_VEL
LIN {X 0,Y 192.265,Z 393.076,A -85,B 0,C 180,E1 -24620.141,E2 -24620.141} C_VEL
LIN {X 0,Y 198.631,Z 380.578,A -85,B 0,C 180,E1 -24621.52,E2 -24621.52} C_VEL
LIN {X 0,Y 203.636,Z 368.096,A -85,B 0,C 180,E1 -24622.54,E2 -24622.54} C_VEL
LIN {X 0,Y 208.02,Z 353.813,A -85,B 0,C 180,E1 -24623.38,E2 -24623.38} C_VEL
LIN {X 0,Y 210.932,Z 339.804,A -85,B 0,C 180,E1 -24623.949,E2 -24623.949} C_VEL
LIN {X 0,Y 212.246,Z 330.731,A -85,B 0,C 180,E1 -24624.294,E2 -24624.294} C_VEL
LIN {X 0,Y 211.177,Z 325.785,A -85,B 0,C 180,E1 -24626.5,E2 -24626.5} C_VEL
LIN {X 0,Y 210.605,Z 323.063,A -85,B 0,C 180,E1 -24628.024,E2 -24628.024} C_VEL
LIN {X 0,Y 210.072,Z 320.498,A -85,B 0,C 180,E1 -24629.879,E2 -24629.879} C_VEL
LIN {X 0,Y 209.603,Z 317.769,A -85,B 0,C 180,E1 -24633.133,E2 -24633.133} C_VEL
LIN {X 0,Y 209.766,Z 316.868,A -85,B 0,C 180,E1 -24636.294,E2 -24636.294} C_VEL
LIN {X 0,Y 210.362,Z 317.151,A -85,B 0,C 180,E1 -24638.859,E2 -24638.859} C_VEL
LIN {X 0,Y 211.651,Z 320.133,A -85,B 0,C 180,E1 -24642.178,E2 -24642.178} C_VEL
LIN {X 0,Y 213.013,Z 323.313,A -85,B 0,C 180,E1 -24644.483,E2 -24644.483} C_VEL
LIN {X 0,Y 213.079,Z 323.527,A -85,B 0,C 180,E1 -24644.594,E2 -24644.594} C_VEL
LIN {X 0,Y 210.268,Z 340.859,A -85,B 0,C 180,E1 -24645.338,E2 -24645.338} C_VEL
LIN {X 0,Y 207.309,Z 352.693,A -85,B 0,C 180,E1 -24646.12,E2 -24646.12} C_VEL
LIN {X 0,Y 202.748,Z 366.038,A -85,B 0,C 180,E1 -24647.319,E2 -24647.319} C_VEL
LIN {X 0,Y 197.613,Z 377.766,A -85,B 0,C 180,E1 -24648.72,E2 -24648.72} C_VEL
LIN {X 0,Y 191.843,Z 388.383,A -85,B 0,C 180,E1 -24650.363,E2 -24650.363} C_VEL
LIN {X 0,Y 185.113,Z 398.723,A -85,B 0,C 180,E1 -24652.492,E2 -24652.492} C_VEL
LIN {X 0,Y 178.18,Z 407.552,A -85,B 0,C 180,E1 -24654.908,E2 -24654.908} C_VEL
LIN {X 0,Y 171.342,Z 415.09,A -85,B 0,C 180,E1 -24657.649,E2 -24657.649} C_VEL
LIN {X 0,Y 166.204,Z 420.003,A -85,B 0,C 180,E1 -24660,E2 -24660} C_VEL
LIN {X 0,Y 159.013,Z 425.907,A -85,B 0,C 180,E1 -24663.801,E2 -24663.801} C_VEL
LIN {X 0,Y 152.593,Z 430.187,A -85,B 0,C 180,E1 -24667.942,E2 -24667.942} C_VEL
LIN {X 0,Y 148.807,Z 432.255,A -85,B 0,C 180,E1 -24670.889,E2 -24670.889} C_VEL
LIN {X 0,Y 145.059,Z 433.826,A -85,B 0,C 180,E1 -24674.309,E2 -24674.309} C_VEL
LIN {X 0,Y 141.102,Z 434.803,A -85,B 0,C 180,E1 -24678.855,E2 -24678.855} C_VEL
LIN {X 0,Y 137.741,Z 434.62,A -85,B 0,C 180,E1 -24684.091,E2 -24684.091} C_VEL
LIN {X 0,Y 135.786,Z 433.513,A -85,B 0,C 180,E1 -24688.373,E2 -24688.373} C_VEL
LIN {X 0,Y 134.419,Z 431.295,A -85,B 0,C 180,E1 -24693.224,E2 -24693.224} C_VEL
LIN {X 0,Y 133.836,Z 428.057,A -85,B 0,C 180,E1 -24698.032,E2 -24698.032} C_VEL
LIN {X 0,Y 134.079,Z 423.567,A -85,B 0,C 180,E1 -24702.954,E2 -24702.954} C_VEL
LIN {X 0,Y 135.024,Z 417.375,A -85,B 0,C 180,E1 -24708.079,E2 -24708.079} C_VEL
LIN {X 0,Y 136.246,Z 410.739,A -85,B 0,C 180,E1 -24712.362,E2 -24712.362} C_VEL
LIN {X 0,Y 138.051,Z 402.345,A -85,B 0,C 180,E1 -24716.682,E2 -24716.682} C_VEL
LIN {X 0,Y 140.421,Z 392.424,A -85,B 0,C 180,E1 -24720.695,E2 -24720.695} C_VEL
LIN {X 0,Y 142.789,Z 381.775,A -85,B 0,C 180,E1 -24724.079,E2 -24724.079} C_VEL
LIN {X 0,Y 145.174,Z 370.483,A -85,B 0,C 180,E1 -24726.898,E2 -24726.898} C_VEL
LIN {X 0,Y 147.378,Z 358.315,A -85,B 0,C 180,E1 -24729.227,E2 -24729.227} C_VEL
LIN {X 0,Y 149.386,Z 345.016,A -85,B 0,C 180,E1 -24731.13,E2 -24731.13} C_VEL
LIN {X 0,Y 150.711,Z 331.453,A -85,B 0,C 180,E1 -24732.488,E2 -24732.488} C_VEL
LIN {X 0,Y 152.529,Z 305.311,A -85,B 0,C 180,E1 -24734.064,E2 -24734.064} C_VEL
LIN {X 0,Y 154.345,Z 279.33,A -85,B 0,C 180,E1 -24735.497,E2 -24735.497} C_VEL
LIN {X 0,Y 145.389,Z 257.117,A -85,B 0,C 180,E1 -24738.648,E2 -24738.648} C_VEL
LIN {X 0,Y 137.748,Z 240.57,A -85,B 0,C 180,E1 -24741.52,E2 -24741.52} C_VEL
LIN {X 0,Y 136.668,Z 238.092,A -85,B 0,C 180,E1 -24741.964,E2 -24741.964} C_VEL
LIN {X 0,Y 136.574,Z 237.473,A -85,B 0,C 180,E1 -24742.051,E2 -24742.051} C_VEL
LIN {X 0,Y 137.13,Z 237.402,A -85,B 0,C 180,E1 -24750.001,E2 -24750.001} C_VEL
LIN {X 0,Y 136.55,Z 237.474,A -85,B 0,C 180,E1 -24758.883,E2 -24758.883} C_VEL
LIN {X 0,Y 136.442,Z 237.488,A -85,B 0,C 180,E1 -24761.891,E2 -24761.891} C_VEL
LIN {X 0,Y 136.243,Z 237.509,A -85,B 0,C 180,E1 -24768.03,E2 -24768.03} C_VEL
LIN {X 0,Y 136.197,Z 237.497,A -85,B 0,C 180,E1 -24771.747,E2 -24771.747} C_VEL
LIN {X 0,Y 136.093,Z 237.532,A -85,B 0,C 180,E1 -24778.611,E2 -24778.611} C_VEL
LIN {X 0,Y 136.041,Z 237.519,A -85,B 0,C 180,E1 -24784.631,E2 -24784.631} C_VEL
LIN {X 0,Y 136.025,Z 237.506,A -85,B 0,C 180,E1 -24789.195,E2 -24789.195} C_VEL
LIN {X 0,Y 135.979,Z 237.538,A -85,B 0,C 180,E1 -24793.649,E2 -24793.649} C_VEL
LIN {X 0,Y 135.984,Z 237.546,A -85,B 0,C 180,E1 -24797.788,E2 -24797.788} C_VEL
LIN {X 0,Y 136.022,Z 237.532,A -85,B 0,C 180,E1 -24801.683,E2 -24801.683} C_VEL
LIN {X 0,Y 136.054,Z 237.534,A -85,B 0,C 180,E1 -24805.742,E2 -24805.742} C_VEL
LIN {X 0,Y 136.141,Z 237.521,A -85,B 0,C 180,E1 -24812.315,E2 -24812.315} C_VEL
LIN {X 0,Y 136.243,Z 237.512,A -85,B 0,C 180,E1 -24818.833,E2 -24818.833} C_VEL
LIN {X 0,Y 136.247,Z 237.499,A -85,B 0,C 180,E1 -24825.054,E2 -24825.054} C_VEL
LIN {X 0,Y 136.428,Z 237.456,A -85,B 0,C 180,E1 -24828.178,E2 -24828.178} C_VEL
LIN {X 0,Y 136.539,Z 237.435,A -85,B 0,C 180,E1 -24831.117,E2 -24831.117} C_VEL
LIN {X 0,Y 137.116,Z 237.405,A -85,B 0,C 180,E1 -24840,E2 -24840} C_VEL
LIN {X 0,Y 136.54,Z 237.452,A -85,B 0,C 180,E1 -24848.883,E2 -24848.883} C_VEL
LIN {X 0,Y 136.417,Z 237.485,A -85,B 0,C 180,E1 -24851.893,E2 -24851.893} C_VEL
LIN {X 0,Y 136.173,Z 237.52,A -85,B 0,C 180,E1 -24858.039,E2 -24858.039} C_VEL
LIN {X 0,Y 136.15,Z 237.511,A -85,B 0,C 180,E1 -24861.694,E2 -24861.694} C_VEL
LIN {X 0,Y 136.09,Z 237.532,A -85,B 0,C 180,E1 -24868.605,E2 -24868.605} C_VEL
LIN {X 0,Y 136.042,Z 237.538,A -85,B 0,C 180,E1 -24874.63,E2 -24874.63} C_VEL
LIN {X 0,Y 136.027,Z 237.543,A -85,B 0,C 180,E1 -24879.194,E2 -24879.194} C_VEL
LIN {X 0,Y 136.109,Z 237.688,A -85,B 0,C 180,E1 -24882.959,E2 -24882.959} C_VEL
LIN {X 0,Y 136.734,Z 240.463,A -85,B 0,C 180,E1 -24884.766,E2 -24884.766} C_VEL
LIN {X 0,Y 143.922,Z 258.996,A -85,B 0,C 180,E1 -24887.737,E2 -24887.737} C_VEL
LIN {X 0,Y 150.26,Z 278.013,A -85,B 0,C 180,E1 -24890.253,E2 -24890.253} C_VEL
LIN {X 0,Y 152.744,Z 313.54,A -85,B 0,C 180,E1 -24893.056,E2 -24893.056} C_VEL
LIN {X 0,Y 150.143,Z 352.007,A -85,B 0,C 180,E1 -24895.317,E2 -24895.317} C_VEL
LIN {X 0,Y 148.63,Z 365.754,A -85,B 0,C 180,E1 -24896.653,E2 -24896.653} C_VEL
LIN {X 0,Y 146.736,Z 377.121,A -85,B 0,C 180,E1 -24898.206,E2 -24898.206} C_VEL
LIN {X 0,Y 144.341,Z 389.307,A -85,B 0,C 180,E1 -24900.462,E2 -24900.462} C_VEL
LIN {X 0,Y 141.845,Z 400.61,A -85,B 0,C 180,E1 -24903.195,E2 -24903.195} C_VEL
LIN {X 0,Y 139.546,Z 410.434,A -85,B 0,C 180,E1 -24906.239,E2 -24906.239} C_VEL
LIN {X 0,Y 137.437,Z 419.546,A -85,B 0,C 180,E1 -24909.807,E2 -24909.807} C_VEL
LIN {X 0,Y 135.74,Z 428.475,A -85,B 0,C 180,E1 -24914.226,E2 -24914.226} C_VEL
LIN {X 0,Y 134.696,Z 435.545,A -85,B 0,C 180,E1 -24918.716,E2 -24918.716} C_VEL
LIN {X 0,Y 134.464,Z 441.157,A -85,B 0,C 180,E1 -24923.252,E2 -24923.252} C_VEL
LIN {X 0,Y 134.533,Z 444.82,A -85,B 0,C 180,E1 -24927.005,E2 -24927.005} C_VEL
LIN {X 0,Y 134.795,Z 447.117,A -85,B 0,C 180,E1 -24929.999,E2 -24929.999} C_VEL
LIN {X 0,Y 134.093,Z 449.796,A -85,B 0,C 180,E1 -24935.239,E2 -24935.239} C_VEL
LIN {X 0,Y 134.031,Z 450.963,A -85,B 0,C 180,E1 -24939.05,E2 -24939.05} C_VEL
LIN {X 0,Y 135.101,Z 451.549,A -85,B 0,C 180,E1 -24945.075,E2 -24945.075} C_VEL
LIN {X 0,Y 137.799,Z 450.707,A -85,B 0,C 180,E1 -24950.916,E2 -24950.916} C_VEL
LIN {X 0,Y 141.989,Z 448.431,A -85,B 0,C 180,E1 -24956.453,E2 -24956.453} C_VEL
LIN {X 0,Y 144.708,Z 446.591,A -85,B 0,C 180,E1 -24959.246,E2 -24959.246} C_VEL
LIN {X 0,Y 146.484,Z 444.983,A -85,B 0,C 180,E1 -24961.375,E2 -24961.375} C_VEL
LIN {X 0,Y 148.279,Z 442.095,A -85,B 0,C 180,E1 -24965.004,E2 -24965.004} C_VEL
LIN {X 0,Y 150.653,Z 438.635,A -85,B 0,C 180,E1 -24968.429,E2 -24968.429} C_VEL
LIN {X 0,Y 153.232,Z 436.115,A -85,B 0,C 180,E1 -24970.179,E2 -24970.179} C_VEL
LIN {X 0,Y 160.664,Z 429.489,A -85,B 0,C 180,E1 -24973.547,E2 -24973.547} C_VEL
LIN {X 0,Y 169.143,Z 420.887,A -85,B 0,C 180,E1 -24976.646,E2 -24976.646} C_VEL
LIN {X 0,Y 176.915,Z 411.748,A -85,B 0,C 180,E1 -24979.005,E2 -24979.005} C_VEL
LIN {X 0,Y 184.349,Z 401.416,A -85,B 0,C 180,E1 -24980.964,E2 -24980.964} C_VEL
LIN {X 0,Y 191.481,Z 389.836,A -85,B 0,C 180,E1 -24982.533,E2 -24982.533} C_VEL
LIN {X 0,Y 197.339,Z 378.275,A -85,B 0,C 180,E1 -24983.683,E2 -24983.683} C_VEL
LIN {X 0,Y 202.226,Z 366.29,A -85,B 0,C 180,E1 -24984.583,E2 -24984.583} C_VEL
LIN {X 0,Y 205.979,Z 354.47,A -85,B 0,C 180,E1 -24985.245,E2 -24985.245} C_VEL
LIN {X 0,Y 209.052,Z 340.751,A -85,B 0,C 180,E1 -24985.794,E2 -24985.794} C_VEL
LIN {X 0,Y 209.985,Z 334.691,A -85,B 0,C 180,E1 -24986.042,E2 -24986.042} C_VEL
LIN {X 0,Y 209.191,Z 330.045,A -85,B 0,C 180,E1 -24988.365,E2 -24988.365} C_VEL
LIN {X 0,Y 208.667,Z 327.109,A -85,B 0,C 180,E1 -24990.458,E2 -24990.458} C_VEL
LIN {X 0,Y 208.364,Z 324.555,A -85,B 0,C 180,E1 -24993.638,E2 -24993.638} C_VEL
LIN {X 0,Y 208.531,Z 323.877,A -85,B 0,C 180,E1 -24996.144,E2 -24996.144} C_VEL
LIN {X 0,Y 209.102,Z 324.27,A -85,B 0,C 180,E1 -24998.806,E2 -24998.806} C_VEL
LIN {X 0,Y 210.258,Z 327.108,A -85,B 0,C 180,E1 -25001.91,E2 -25001.91} C_VEL
LIN {X 0,Y 210.725,Z 328.355,A -85,B 0,C 180,E1 -25002.88,E2 -25002.88} C_VEL
LIN {X 0,Y 208.255,Z 342.422,A -85,B 0,C 180,E1 -25003.524,E2 -25003.524} C_VEL
LIN {X 0,Y 205.258,Z 353.766,A -85,B 0,C 180,E1 -25004.258,E2 -25004.258} C_VEL
LIN {X 0,Y 200.709,Z 366.603,A -85,B 0,C 180,E1 -25005.384,E2 -25005.384} C_VEL
LIN {X 0,Y 195.232,Z 378.499,A -85,B 0,C 180,E1 -25006.756,E2 -25006.756} C_VEL
LIN {X 0,Y 188.821,Z 389.664,A -85,B 0,C 180,E1 -25008.459,E2 -25008.459} C_VEL
LIN {X 0,Y 181.844,Z 399.852,A -85,B 0,C 180,E1 -25010.545,E2 -25010.545} C_VEL
LIN {X 0,Y 174.258,Z 409.021,A -85,B 0,C 180,E1 -25013.05,E2 -25013.05} C_VEL
LIN {X 0,Y 167.07,Z 416.382,A -85,B 0,C 180,E1 -25015.778,E2 -25015.778} C_VEL
LIN {X 0,Y 159.993,Z 422.515,A -85,B 0,C 180,E1 -25018.892,E2 -25018.892} C_VEL
LIN {X 0,Y 152.842,Z 427.727,A -85,B 0,C 180,E1 -25022.635,E2 -25022.635} C_VEL
LIN {X 0,Y 146.151,Z 431.66,A -85,B 0,C 180,E1 -25026.903,E2 -25026.903} C_VEL
LIN {X 0,Y 140.335,Z 434.181,A -85,B 0,C 180,E1 -25031.556,E2 -25031.556} C_VEL
LIN {X 0,Y 137.009,Z 435.111,A -85,B 0,C 180,E1 -25034.861,E2 -25034.861} C_VEL
LIN {X 0,Y 133.685,Z 435.498,A -85,B 0,C 180,E1 -25038.867,E2 -25038.867} C_VEL
LIN {X 0,Y 130.624,Z 434.953,A -85,B 0,C 180,E1 -25043.845,E2 -25043.845} C_VEL
LIN {X 0,Y 128.208,Z 433.094,A -85,B 0,C 180,E1 -25049.561,E2 -25049.561} C_VEL
LIN {X 0,Y 126.942,Z 429.695,A -85,B 0,C 180,E1 -25055.667,E2 -25055.667} C_VEL
LIN {X 0,Y 126.856,Z 424.764,A -85,B 0,C 180,E1 -25061.668,E2 -25061.668} C_VEL
LIN {X 0,Y 127.724,Z 418.517,A -85,B 0,C 180,E1 -25067.317,E2 -25067.317} C_VEL
LIN {X 0,Y 128.863,Z 412.337,A -85,B 0,C 180,E1 -25071.67,E2 -25071.67} C_VEL
LIN {X 0,Y 130.776,Z 403.516,A -85,B 0,C 180,E1 -25076.576,E2 -25076.576} C_VEL
LIN {X 0,Y 133.046,Z 394.222,A -85,B 0,C 180,E1 -25080.644,E2 -25080.644} C_VEL
LIN {X 0,Y 135.492,Z 383.697,A -85,B 0,C 180,E1 -25084.253,E2 -25084.253} C_VEL
LIN {X 0,Y 138.027,Z 372.296,A -85,B 0,C 180,E1 -25087.31,E2 -25087.31} C_VEL
LIN {X 0,Y 140.326,Z 360.157,A -85,B 0,C 180,E1 -25089.822,E2 -25089.822} C_VEL
LIN {X 0,Y 142.292,Z 347.964,A -85,B 0,C 180,E1 -25091.711,E2 -25091.711} C_VEL
LIN {X 0,Y 143.879,Z 334.122,A -85,B 0,C 180,E1 -25093.26,E2 -25093.26} C_VEL
LIN {X 0,Y 145.294,Z 315.437,A -85,B 0,C 180,E1 -25094.518,E2 -25094.518} C_VEL
LIN {X 0,Y 147.698,Z 280.73,A -85,B 0,C 180,E1 -25096.532,E2 -25096.532} C_VEL
LIN {X 0,Y 139.036,Z 259.194,A -85,B 0,C 180,E1 -25099.81,E2 -25099.81} C_VEL
LIN {X 0,Y 132.173,Z 244.355,A -85,B 0,C 180,E1 -25102.525,E2 -25102.525} C_VEL
LIN {X 0,Y 129.605,Z 239.039,A -85,B 0,C 180,E1 -25103.614,E2 -25103.614} C_VEL
LIN {X 0,Y 129.5,Z 238.353,A -85,B 0,C 180,E1 -25103.77,E2 -25103.77} C_VEL
LIN {X 0,Y 130.085,Z 238.28,A -85,B 0,C 180,E1 -25110.001,E2 -25110.001} C_VEL
LIN {X 0,Y 129.476,Z 238.355,A -85,B 0,C 180,E1 -25119.373,E2 -25119.373} C_VEL
LIN {X 0,Y 129.345,Z 238.373,A -85,B 0,C 180,E1 -25122.554,E2 -25122.554} C_VEL
LIN {X 0,Y 129.154,Z 238.387,A -85,B 0,C 180,E1 -25129.057,E2 -25129.057} C_VEL
LIN {X 0,Y 129.109,Z 238.38,A -85,B 0,C 180,E1 -25132.399,E2 -25132.399} C_VEL
LIN {X 0,Y 129.018,Z 238.415,A -85,B 0,C 180,E1 -25139.359,E2 -25139.359} C_VEL
LIN {X 0,Y 128.956,Z 238.395,A -85,B 0,C 180,E1 -25145.166,E2 -25145.166} C_VEL
LIN {X 0,Y 128.924,Z 238.401,A -85,B 0,C 180,E1 -25150.857,E2 -25150.857} C_VEL
LIN {X 0,Y 128.913,Z 238.423,A -85,B 0,C 180,E1 -25155.133,E2 -25155.133} C_VEL
LIN {X 0,Y 128.935,Z 238.421,A -85,B 0,C 180,E1 -25159.741,E2 -25159.741} C_VEL
LIN {X 0,Y 128.957,Z 238.413,A -85,B 0,C 180,E1 -25164.835,E2 -25164.835} C_VEL
LIN {X 0,Y 129.019,Z 238.413,A -85,B 0,C 180,E1 -25170.643,E2 -25170.643} C_VEL
LIN {X 0,Y 129.11,Z 238.399,A -85,B 0,C 180,E1 -25177.602,E2 -25177.602} C_VEL
LIN {X 0,Y 129.15,Z 238.396,A -85,B 0,C 180,E1 -25180.944,E2 -25180.944} C_VEL
LIN {X 0,Y 129.349,Z 238.338,A -85,B 0,C 180,E1 -25187.965,E2 -25187.965} C_VEL
LIN {X 0,Y 129.465,Z 238.313,A -85,B 0,C 180,E1 -25190.628,E2 -25190.628} C_VEL
LIN {X 0,Y 130.071,Z 238.283,A -85,B 0,C 180,E1 -25200,E2 -25200} C_VEL
LIN {X 0,Y 129.465,Z 238.335,A -85,B 0,C 180,E1 -25209.373,E2 -25209.373} C_VEL
LIN {X 0,Y 129.301,Z 238.375,A -85,B 0,C 180,E1 -25212.558,E2 -25212.558} C_VEL
LIN {X 0,Y 129.089,Z 238.398,A -85,B 0,C 180,E1 -25219.066,E2 -25219.066} C_VEL
LIN {X 0,Y 129.046,Z 238.399,A -85,B 0,C 180,E1 -25222.41,E2 -25222.41} C_VEL
LIN {X 0,Y 129.019,Z 238.407,A -85,B 0,C 180,E1 -25229.358,E2 -25229.358} C_VEL
LIN {X 0,Y 128.958,Z 238.42,A -85,B 0,C 180,E1 -25235.165,E2 -25235.165} C_VEL
LIN {X 0,Y 129.027,Z 238.562,A -85,B 0,C 180,E1 -25241.987,E2 -25241.987} C_VEL
LIN {X 0,Y 129.362,Z 239.91,A -85,B 0,C 180,E1 -25242.907,E2 -25242.907} C_VEL
LIN {X 0,Y 135.822,Z 256.122,A -85,B 0,C 180,E1 -25245.784,E2 -25245.784} C_VEL
LIN {X 0,Y 141.865,Z 273.571,A -85,B 0,C 180,E1 -25248.396,E2 -25248.396} C_VEL
LIN {X 0,Y 143.951,Z 280.671,A -85,B 0,C 180,E1 -25249.312,E2 -25249.312} C_VEL
LIN {X 0,Y 146.129,Z 314.55,A -85,B 0,C 180,E1 -25252.092,E2 -25252.092} C_VEL
LIN {X 0,Y 143.502,Z 351.12,A -85,B 0,C 180,E1 -25254.33,E2 -25254.33} C_VEL
LIN {X 0,Y 141.967,Z 364.955,A -85,B 0,C 180,E1 -25255.728,E2 -25255.728} C_VEL
LIN {X 0,Y 140.007,Z 376.383,A -85,B 0,C 180,E1 -25257.341,E2 -25257.341} C_VEL
LIN {X 0,Y 137.534,Z 388.619,A -85,B 0,C 180,E1 -25259.694,E2 -25259.694} C_VEL
LIN {X 0,Y 134.903,Z 400.202,A -85,B 0,C 180,E1 -25262.622,E2 -25262.622} C_VEL
LIN {X 0,Y 132.6,Z 409.811,A -85,B 0,C 180,E1 -25265.746,E2 -25265.746} C_VEL
LIN {X 0,Y 130.411,Z 418.932,A -85,B 0,C 180,E1 -25269.494,E2 -25269.494} C_VEL
LIN {X 0,Y 128.673,Z 427.872,A -85,B 0,C 180,E1 -25274.151,E2 -25274.151} C_VEL
LIN {X 0,Y 127.627,Z 434.955,A -85,B 0,C 180,E1 -25278.887,E2 -25278.887} C_VEL
LIN {X 0,Y 127.44,Z 440.567,A -85,B 0,C 180,E1 -25283.667,E2 -25283.667} C_VEL
LIN {X 0,Y 127.595,Z 444.829,A -85,B 0,C 180,E1 -25288.421,E2 -25288.421} C_VEL
LIN {X 0,Y 127.759,Z 446.005,A -85,B 0,C 180,E1 -25289.999,E2 -25289.999} C_VEL
LIN {X 0,Y 127.064,Z 448.786,A -85,B 0,C 180,E1 -25295.378,E2 -25295.378} C_VEL
LIN {X 0,Y 127.021,Z 450.106,A -85,B 0,C 180,E1 -25299.554,E2 -25299.554} C_VEL
LIN {X 0,Y 128.225,Z 450.952,A -85,B 0,C 180,E1 -25305.905,E2 -25305.905} C_VEL
LIN {X 0,Y 131.175,Z 450.315,A -85,B 0,C 180,E1 -25312.026,E2 -25312.026} C_VEL
LIN {X 0,Y 135.627,Z 448.256,A -85,B 0,C 180,E1 -25317.798,E2 -25317.798} C_VEL
LIN {X 0,Y 138.351,Z 446.685,A -85,B 0,C 180,E1 -25320.529,E2 -25320.529} C_VEL
LIN {X 0,Y 143.186,Z 443.592,A -85,B 0,C 180,E1 -25324.363,E2 -25324.363} C_VEL
LIN {X 0,Y 148.824,Z 439.582,A -85,B 0,C 180,E1 -25327.872,E2 -25327.872} C_VEL
LIN {X 0,Y 153.232,Z 436.115,A -85,B 0,C 180,E1 -25330.179,E2 -25330.179} C_VEL
LIN {X 0,Y 155.955,Z 433.461,A -85,B 0,C 180,E1 -25331.853,E2 -25331.853} C_VEL
LIN {X 0,Y 159.282,Z 428.996,A -85,B 0,C 180,E1 -25334.848,E2 -25334.848} C_VEL
LIN {X 0,Y 162.896,Z 424.097,A -85,B 0,C 180,E1 -25337.611,E2 -25337.611} C_VEL
LIN {X 0,Y 165.941,Z 420.674,A -85,B 0,C 180,E1 -25338.897,E2 -25338.897} C_VEL
LIN {X 0,Y 173.792,Z 411.919,A -85,B 0,C 180,E1 -25341.119,E2 -25341.119} C_VEL
LIN {X 0,Y 181.508,Z 401.882,A -85,B 0,C 180,E1 -25342.996,E2 -25342.996} C_VEL
LIN {X 0,Y 188.829,Z 390.587,A -85,B 0,C 180,E1 -25344.504,E2 -25344.504} C_VEL
LIN {X 0,Y 194.843,Z 379.417,A -85,B 0,C 180,E1 -25345.598,E2 -25345.598} C_VEL
LIN {X 0,Y 200.156,Z 367.039,A -85,B 0,C 180,E1 -25346.503,E2 -25346.503} C_VEL
LIN {X 0,Y 204.671,Z 353.404,A -85,B 0,C 180,E1 -25347.219,E2 -25347.219} C_VEL
LIN {X 0,Y 207.873,Z 339.29,A -85,B 0,C 180,E1 -25347.762,E2 -25347.762} C_VEL
LIN {X 0,Y 207.885,Z 338.549,A -85,B 0,C 180,E1 -25347.985,E2 -25347.985} C_VEL
LIN {X 0,Y 207.594,Z 335.861,A -85,B 0,C 180,E1 -25349.481,E2 -25349.481} C_VEL
LIN {X 0,Y 207.266,Z 333.551,A -85,B 0,C 180,E1 -25351.246,E2 -25351.246} C_VEL
LIN {X 0,Y 207.14,Z 331.522,A -85,B 0,C 180,E1 -25353.827,E2 -25353.827} C_VEL
LIN {X 0,Y 207.336,Z 330.865,A -85,B 0,C 180,E1 -25356.234,E2 -25356.234} C_VEL
LIN {X 0,Y 207.802,Z 331.246,A -85,B 0,C 180,E1 -25358.552,E2 -25358.552} C_VEL
LIN {X 0,Y 208.644,Z 333.464,A -85,B 0,C 180,E1 -25361.132,E2 -25361.132} C_VEL
LIN {X 0,Y 205.848,Z 346.72,A -85,B 0,C 180,E1 -25361.807,E2 -25361.807} C_VEL
LIN {X 0,Y 201.943,Z 359.415,A -85,B 0,C 180,E1 -25362.721,E2 -25362.721} C_VEL
LIN {X 0,Y 197.223,Z 371.026,A -85,B 0,C 180,E1 -25363.8,E2 -25363.8} C_VEL
LIN {X 0,Y 191.652,Z 382.05,A -85,B 0,C 180,E1 -25365.126,E2 -25365.126} C_VEL
LIN {X 0,Y 186.062,Z 391.156,A -85,B 0,C 180,E1 -25366.514,E2 -25366.514} C_VEL
LIN {X 0,Y 178.45,Z 401.508,A -85,B 0,C 180,E1 -25368.643,E2 -25368.643} C_VEL
LIN {X 0,Y 170.17,Z 410.865,A -85,B 0,C 180,E1 -25371.227,E2 -25371.227} C_VEL
LIN {X 0,Y 162.54,Z 418.08,A -85,B 0,C 180,E1 -25373.977,E2 -25373.977} C_VEL
LIN {X 0,Y 154.491,Z 424.457,A -85,B 0,C 180,E1 -25377.392,E2 -25377.392} C_VEL
LIN {X 0,Y 147.603,Z 428.965,A -85,B 0,C 180,E1 -25380.861,E2 -25380.861} C_VEL
LIN {X 0,Y 141.063,Z 432.466,A -85,B 0,C 180,E1 -25384.847,E2 -25384.847} C_VEL
LIN {X 0,Y 135.267,Z 434.759,A -85,B 0,C 180,E1 -25389.192,E2 -25389.192} C_VEL
LIN {X 0,Y 130.32,Z 435.931,A -85,B 0,C 180,E1 -25393.903,E2 -25393.903} C_VEL
LIN {X 0,Y 125.794,Z 435.945,A -85,B 0,C 180,E1 -25399.585,E2 -25399.585} C_VEL
LIN {X 0,Y 123.204,Z 435.066,A -85,B 0,C 180,E1 -25404.121,E2 -25404.121} C_VEL
LIN {X 0,Y 121.087,Z 433.069,A -85,B 0,C 180,E1 -25409.472,E2 -25409.472} C_VEL
LIN {X 0,Y 119.823,Z 429.329,A -85,B 0,C 180,E1 -25415.911,E2 -25415.911} C_VEL
LIN {X 0,Y 119.817,Z 423.947,A -85,B 0,C 180,E1 -25422.419,E2 -25422.419} C_VEL
LIN {X 0,Y 120.78,Z 417.627,A -85,B 0,C 180,E1 -25428.067,E2 -25428.067} C_VEL
LIN {X 0,Y 122.037,Z 411.036,A -85,B 0,C 180,E1 -25432.721,E2 -25432.721} C_VEL
LIN {X 0,Y 124.001,Z 402.52,A -85,B 0,C 180,E1 -25437.52,E2 -25437.52} C_VEL
LIN {X 0,Y 126.535,Z 392.471,A -85,B 0,C 180,E1 -25441.923,E2 -25441.923} C_VEL
LIN {X 0,Y 128.955,Z 382.303,A -85,B 0,C 180,E1 -25445.445,E2 -25445.445} C_VEL
LIN {X 0,Y 131.38,Z 371.637,A -85,B 0,C 180,E1 -25448.359,E2 -25448.359} C_VEL
LIN {X 0,Y 133.809,Z 359.141,A -85,B 0,C 180,E1 -25450.98,E2 -25450.98} C_VEL
LIN {X 0,Y 135.798,Z 347.035,A -85,B 0,C 180,E1 -25452.883,E2 -25452.883} C_VEL
LIN {X 0,Y 137.403,Z 333.164,A -85,B 0,C 180,E1 -25454.425,E2 -25454.425} C_VEL
LIN {X 0,Y 139.015,Z 310.938,A -85,B 0,C 180,E1 -25455.932,E2 -25455.932} C_VEL
LIN {X 0,Y 141.125,Z 282.34,A -85,B 0,C 180,E1 -25457.648,E2 -25457.648} C_VEL
LIN {X 0,Y 133.403,Z 262.934,A -85,B 0,C 180,E1 -25460.733,E2 -25460.733} C_VEL
LIN {X 0,Y 126.626,Z 247.996,A -85,B 0,C 180,E1 -25463.628,E2 -25463.628} C_VEL
LIN {X 0,Y 122.721,Z 240.3,A -85,B 0,C 180,E1 -25465.382,E2 -25465.382} C_VEL
LIN {X 0,Y 122.515,Z 239.223,A -85,B 0,C 180,E1 -25465.683,E2 -25465.683} C_VEL
LIN {X 0,Y 123.038,Z 239.158,A -85,B 0,C 180,E1 -25470.001,E2 -25470.001} C_VEL
LIN {X 0,Y 122.419,Z 239.234,A -85,B 0,C 180,E1 -25476.594,E2 -25476.594} C_VEL
LIN {X 0,Y 122.319,Z 239.249,A -85,B 0,C 180,E1 -25482.377,E2 -25482.377} C_VEL
LIN {X 0,Y 122.109,Z 239.273,A -85,B 0,C 180,E1 -25486.726,E2 -25486.726} C_VEL
LIN {X 0,Y 122.028,Z 239.262,A -85,B 0,C 180,E1 -25492.855,E2 -25492.855} C_VEL
LIN {X 0,Y 121.94,Z 239.294,A -85,B 0,C 180,E1 -25497.458,E2 -25497.458} C_VEL
LIN {X 0,Y 121.899,Z 239.298,A -85,B 0,C 180,E1 -25501.259,E2 -25501.259} C_VEL
LIN {X 0,Y 121.881,Z 239.267,A -85,B 0,C 180,E1 -25506.169,E2 -25506.169} C_VEL
LIN {X 0,Y 121.864,Z 239.283,A -85,B 0,C 180,E1 -25511.434,E2 -25511.434} C_VEL
LIN {X 0,Y 121.864,Z 239.304,A -85,B 0,C 180,E1 -25518.567,E2 -25518.567} C_VEL
LIN {X 0,Y 121.909,Z 239.29,A -85,B 0,C 180,E1 -25524.796,E2 -25524.796} C_VEL
LIN {X 0,Y 121.928,Z 239.296,A -85,B 0,C 180,E1 -25529.84,E2 -25529.84} C_VEL
LIN {X 0,Y 121.983,Z 239.281,A -85,B 0,C 180,E1 -25536.215,E2 -25536.215} C_VEL
LIN {X 0,Y 122.044,Z 239.28,A -85,B 0,C 180,E1 -25539.787,E2 -25539.787} C_VEL
LIN {X 0,Y 122.099,Z 239.268,A -85,B 0,C 180,E1 -25543.274,E2 -25543.274} C_VEL
LIN {X 0,Y 122.394,Z 239.192,A -85,B 0,C 180,E1 -25550.081,E2 -25550.081} C_VEL
LIN {X 0,Y 122.589,Z 239.207,A -85,B 0,C 180,E1 -25556.714,E2 -25556.714} C_VEL
LIN {X 0,Y 123.025,Z 239.16,A -85,B 0,C 180,E1 -25560,E2 -25560} C_VEL
LIN {X 0,Y 122.409,Z 239.212,A -85,B 0,C 180,E1 -25566.594,E2 -25566.594} C_VEL
LIN {X 0,Y 122.394,Z 239.218,A -85,B 0,C 180,E1 -25569.92,E2 -25569.92} C_VEL
LIN {X 0,Y 122.19,Z 239.263,A -85,B 0,C 180,E1 -25573.301,E2 -25573.301} C_VEL
LIN {X 0,Y 121.992,Z 239.274,A -85,B 0,C 180,E1 -25580.223,E2 -25580.223} C_VEL
LIN {X 0,Y 121.943,Z 239.292,A -85,B 0,C 180,E1 -25583.793,E2 -25583.793} C_VEL
LIN {X 0,Y 121.928,Z 239.287,A -85,B 0,C 180,E1 -25590.16,E2 -25590.16} C_VEL
LIN {X 0,Y 121.882,Z 239.3,A -85,B 0,C 180,E1 -25596.168,E2 -25596.168} C_VEL
LIN {X 0,Y 121.949,Z 239.428,A -85,B 0,C 180,E1 -25600.84,E2 -25600.84} C_VEL
LIN {X 0,Y 122.986,Z 242.233,A -85,B 0,C 180,E1 -25601.391,E2 -25601.391} C_VEL
LIN {X 0,Y 125.716,Z 248.292,A -85,B 0,C 180,E1 -25602.675,E2 -25602.675} C_VEL
LIN {X 0,Y 132.016,Z 264.785,A -85,B 0,C 180,E1 -25605.609,E2 -25605.609} C_VEL
LIN {X 0,Y 137.602,Z 282.142,A -85,B 0,C 180,E1 -25608.179,E2 -25608.179} C_VEL
LIN {X 0,Y 139.525,Z 315.721,A -85,B 0,C 180,E1 -25611.066,E2 -25611.066} C_VEL
LIN {X 0,Y 136.831,Z 351.166,A -85,B 0,C 180,E1 -25613.337,E2 -25613.337} C_VEL
LIN {X 0,Y 135.353,Z 364.153,A -85,B 0,C 180,E1 -25614.714,E2 -25614.714} C_VEL
LIN {X 0,Y 133.323,Z 375.647,A -85,B 0,C 180,E1 -25616.392,E2 -25616.392} C_VEL
LIN {X 0,Y 131.028,Z 386.691,A -85,B 0,C 180,E1 -25618.558,E2 -25618.558} C_VEL
LIN {X 0,Y 128.495,Z 397.621,A -85,B 0,C 180,E1 -25621.353,E2 -25621.353} C_VEL
LIN {X 0,Y 125.87,Z 408.126,A -85,B 0,C 180,E1 -25624.801,E2 -25624.801} C_VEL
LIN {X 0,Y 123.767,Z 416.64,A -85,B 0,C 180,E1 -25628.339,E2 -25628.339} C_VEL
LIN {X 0,Y 122.106,Z 424.499,A -85,B 0,C 180,E1 -25632.411,E2 -25632.411} C_VEL
LIN {X 0,Y 120.851,Z 432.121,A -85,B 0,C 180,E1 -25637.403,E2 -25637.403} C_VEL
LIN {X 0,Y 120.393,Z 438.699,A -85,B 0,C 180,E1 -25642.925,E2 -25642.925} C_VEL
LIN {X 0,Y 120.563,Z 443.572,A -85,B 0,C 180,E1 -25648.329,E2 -25648.329} C_VEL
LIN {X 0,Y 120.745,Z 444.772,A -85,B 0,C 180,E1 -25649.999,E2 -25649.999} C_VEL
LIN {X 0,Y 120.048,Z 447.715,A -85,B 0,C 180,E1 -25655.59,E2 -25655.59} C_VEL
LIN {X 0,Y 120.023,Z 449.242,A -85,B 0,C 180,E1 -25660.117,E2 -25660.117} C_VEL
LIN {X 0,Y 121.387,Z 450.266,A -85,B 0,C 180,E1 -25666.826,E2 -25666.826} C_VEL
LIN {X 0,Y 124.608,Z 449.904,A -85,B 0,C 180,E1 -25673.253,E2 -25673.253} C_VEL
LIN {X 0,Y 129.35,Z 448.075,A -85,B 0,C 180,E1 -25679.274,E2 -25679.274} C_VEL
LIN {X 0,Y 135.594,Z 444.813,A -85,B 0,C 180,E1 -25684.759,E2 -25684.759} C_VEL
LIN {X 0,Y 141.253,Z 441.339,A -85,B 0,C 180,E1 -25688.457,E2 -25688.457} C_VEL
LIN {X 0,Y 149.849,Z 435.24,A -85,B 0,C 180,E1 -25692.847,E2 -25692.847} C_VEL
LIN {X 0,Y 156.879,Z 429.403,A -85,B 0,C 180,E1 -25695.789,E2 -25695.789} C_VEL
LIN {X 0,Y 164.419,Z 422.255,A -85,B 0,C 180,E1 -25698.419,E2 -25698.419} C_VEL
LIN {X 0,Y 165.941,Z 420.674,A -85,B 0,C 180,E1 -25698.897,E2 -25698.897} C_VEL
LIN {X 0,Y 169.061,Z 417.101,A -85,B 0,C 180,E1 -25700.111,E2 -25700.111} C_VEL
LIN {X 0,Y 173.15,Z 411.24,A -85,B 0,C 180,E1 -25702.427,E2 -25702.427} C_VEL
LIN {X 0,Y 177.23,Z 404.9,A -85,B 0,C 180,E1 -25704.506,E2 -25704.506} C_VEL
LIN {X 0,Y 180.21,Z 400.593,A -85,B 0,C 180,E1 -25705.351,E2 -25705.351} C_VEL
LIN {X 0,Y 187.96,Z 388.873,A -85,B 0,C 180,E1 -25706.784,E2 -25706.784} C_VEL
LIN {X 0,Y 194.136,Z 377.499,A -85,B 0,C 180,E1 -25707.801,E2 -25707.801} C_VEL
LIN {X 0,Y 198.786,Z 366.991,A -85,B 0,C 180,E1 -25708.516,E2 -25708.516} C_VEL
LIN {X 0,Y 203.623,Z 352.876,A -85,B 0,C 180,E1 -25709.22,E2 -25709.22} C_VEL
LIN {X 0,Y 206.035,Z 343.106,A -85,B 0,C 180,E1 -25709.628,E2 -25709.628} C_VEL
LIN {X 0,Y 205.872,Z 340.323,A -85,B 0,C 180,E1 -25711.694,E2 -25711.694} C_VEL
LIN {X 0,Y 205.835,Z 338.382,A -85,B 0,C 180,E1 -25714.235,E2 -25714.235} C_VEL
LIN {X 0,Y 206.162,Z 337.893,A -85,B 0,C 180,E1 -25716.987,E2 -25716.987} C_VEL
LIN {X 0,Y 206.433,Z 338.228,A -85,B 0,C 180,E1 -25718.403,E2 -25718.403} C_VEL
LIN {X 0,Y 206.617,Z 339.147,A -85,B 0,C 180,E1 -25719.461,E2 -25719.461} C_VEL
LIN {X 0,Y 203.742,Z 350.629,A -85,B 0,C 180,E1 -25720.06,E2 -25720.06} C_VEL
LIN {X 0,Y 199.443,Z 363.19,A -85,B 0,C 180,E1 -25720.986,E2 -25720.986} C_VEL
LIN {X 0,Y 194.704,Z 373.881,A -85,B 0,C 180,E1 -25721.997,E2 -25721.997} C_VEL
LIN {X 0,Y 188.985,Z 384.264,A -85,B 0,C 180,E1 -25723.249,E2 -25723.249} C_VEL
LIN {X 0,Y 181.973,Z 394.771,A -85,B 0,C 180,E1 -25724.911,E2 -25724.911} C_VEL
LIN {X 0,Y 174.92,Z 403.678,A -85,B 0,C 180,E1 -25726.768,E2 -25726.768} C_VEL
LIN {X 0,Y 167.21,Z 411.849,A -85,B 0,C 180,E1 -25729.025,E2 -25729.025} C_VEL
LIN {X 0,Y 159.103,Z 419.031,A -85,B 0,C 180,E1 -25731.746,E2 -25731.746} C_VEL
LIN {X 0,Y 151.623,Z 424.655,A -85,B 0,C 180,E1 -25734.681,E2 -25734.681} C_VEL
LIN {X 0,Y 143.229,Z 429.863,A -85,B 0,C 180,E1 -25738.594,E2 -25738.594} C_VEL
LIN {X 0,Y 135.652,Z 433.474,A -85,B 0,C 180,E1 -25742.97,E2 -25742.97} C_VEL
LIN {X 0,Y 131.116,Z 435.117,A -85,B 0,C 180,E1 -25746.154,E2 -25746.154} C_VEL
LIN {X 0,Y 126.978,Z 436.19,A -85,B 0,C 180,E1 -25749.558,E2 -25749.558} C_VEL
LIN {X 0,Y 122.932,Z 436.716,A -85,B 0,C 180,E1 -25753.622,E2 -25753.622} C_VEL
LIN {X 0,Y 118.844,Z 436.382,A -85,B 0,C 180,E1 -25758.885,E2 -25758.885} C_VEL
LIN {X 0,Y 115.447,Z 434.714,A -85,B 0,C 180,E1 -25765.222,E2 -25765.222} C_VEL
LIN {X 0,Y 113.319,Z 431.576,A -85,B 0,C 180,E1 -25771.948,E2 -25771.948} C_VEL
LIN {X 0,Y 112.549,Z 427.051,A -85,B 0,C 180,E1 -25778.641,E2 -25778.641} C_VEL
LIN {X 0,Y 113.078,Z 421.027,A -85,B 0,C 180,E1 -25785.136,E2 -25785.136} C_VEL
LIN {X 0,Y 114.137,Z 415.183,A -85,B 0,C 180,E1 -25790.069,E2 -25790.069} C_VEL
LIN {X 0,Y 115.64,Z 407.985,A -85,B 0,C 180,E1 -25794.935,E2 -25794.935} C_VEL
LIN {X 0,Y 117.773,Z 399.148,A -85,B 0,C 180,E1 -25799.701,E2 -25799.701} C_VEL
LIN {X 0,Y 120.173,Z 390.036,A -85,B 0,C 180,E1 -25803.578,E2 -25803.578} C_VEL
LIN {X 0,Y 122.917,Z 378.947,A -85,B 0,C 180,E1 -25807.299,E2 -25807.299} C_VEL
LIN {X 0,Y 125.563,Z 367.105,A -85,B 0,C 180,E1 -25810.378,E2 -25810.378} C_VEL
LIN {X 0,Y 127.975,Z 354.472,A -85,B 0,C 180,E1 -25812.833,E2 -25812.833} C_VEL
LIN {X 0,Y 129.85,Z 342.11,A -85,B 0,C 180,E1 -25814.609,E2 -25814.609} C_VEL
LIN {X 0,Y 131.234,Z 328.661,A -85,B 0,C 180,E1 -25815.937,E2 -25815.937} C_VEL
LIN {X 0,Y 134.625,Z 283.988,A -85,B 0,C 180,E1 -25818.807,E2 -25818.807} C_VEL
LIN {X 0,Y 127.234,Z 265.334,A -85,B 0,C 180,E1 -25821.989,E2 -25821.989} C_VEL
LIN {X 0,Y 121.062,Z 251.561,A -85,B 0,C 180,E1 -25824.828,E2 -25824.828} C_VEL
LIN {X 0,Y 115.789,Z 241.045,A -85,B 0,C 180,E1 -25827.392,E2 -25827.392} C_VEL
LIN {X 0,Y 115.631,Z 240.08,A -85,B 0,C 180,E1 -25827.606,E2 -25827.606} C_VEL
LIN {X 0,Y 115.99,Z 240.035,A -85,B 0,C 180,E1 -25830.001,E2 -25830.001} C_VEL
LIN {X 0,Y 115.36,Z 240.113,A -85,B 0,C 180,E1 -25837,E2 -25837} C_VEL
LIN {X 0,Y 115.253,Z 240.129,A -85,B 0,C 180,E1 -25842.667,E2 -25842.667} C_VEL
LIN {X 0,Y 115.012,Z 240.154,A -85,B 0,C 180,E1 -25847.791,E2 -25847.791} C_VEL
LIN {X 0,Y 114.947,Z 240.147,A -85,B 0,C 180,E1 -25853.492,E2 -25853.492} C_VEL
LIN {X 0,Y 114.856,Z 240.176,A -85,B 0,C 180,E1 -25861.057,E2 -25861.057} C_VEL
LIN {X 0,Y 114.774,Z 240.144,A -85,B 0,C 180,E1 -25867.76,E2 -25867.76} C_VEL
LIN {X 0,Y 114.779,Z 240.173,A -85,B 0,C 180,E1 -25872.713,E2 -25872.713} C_VEL
LIN {X 0,Y 114.787,Z 240.187,A -85,B 0,C 180,E1 -25877.663,E2 -25877.663} C_VEL
LIN {X 0,Y 114.784,Z 240.174,A -85,B 0,C 180,E1 -25882.748,E2 -25882.748} C_VEL
LIN {X 0,Y 114.857,Z 240.178,A -85,B 0,C 180,E1 -25888.945,E2 -25888.945} C_VEL
LIN {X 0,Y 114.948,Z 240.158,A -85,B 0,C 180,E1 -25896.51,E2 -25896.51} C_VEL
LIN {X 0,Y 115.006,Z 240.156,A -85,B 0,C 180,E1 -25902.209,E2 -25902.209} C_VEL
LIN {X 0,Y 115.309,Z 240.074,A -85,B 0,C 180,E1 -25909.465,E2 -25909.465} C_VEL
LIN {X 0,Y 115.513,Z 240.087,A -85,B 0,C 180,E1 -25916.512,E2 -25916.512} C_VEL
LIN {X 0,Y 115.977,Z 240.038,A -85,B 0,C 180,E1 -25920,E2 -25920} C_VEL
LIN {X 0,Y 115.351,Z 240.087,A -85,B 0,C 180,E1 -25926.999,E2 -25926.999} C_VEL
LIN {X 0,Y 115.207,Z 240.13,A -85,B 0,C 180,E1 -25932.56,E2 -25932.56} C_VEL
LIN {X 0,Y 114.97,Z 240.161,A -85,B 0,C 180,E1 -25937.797,E2 -25937.797} C_VEL
LIN {X 0,Y 114.909,Z 240.167,A -85,B 0,C 180,E1 -25943.445,E2 -25943.445} C_VEL
LIN {X 0,Y 114.857,Z 240.167,A -85,B 0,C 180,E1 -25951.056,E2 -25951.056} C_VEL
LIN {X 0,Y 114.809,Z 240.252,A -85,B 0,C 180,E1 -25958.722,E2 -25958.722} C_VEL
LIN {X 0,Y 115.805,Z 242.97,A -85,B 0,C 180,E1 -25959.304,E2 -25959.304} C_VEL
LIN {X 0,Y 118.346,Z 247.4,A -85,B 0,C 180,E1 -25960.506,E2 -25960.506} C_VEL
LIN {X 0,Y 124.737,Z 263.835,A -85,B 0,C 180,E1 -25963.777,E2 -25963.777} C_VEL
LIN {X 0,Y 131.215,Z 283.654,A -85,B 0,C 180,E1 -25966.957,E2 -25966.957} C_VEL
LIN {X 0,Y 133.032,Z 315.719,A -85,B 0,C 180,E1 -25969.859,E2 -25969.859} C_VEL
LIN {X 0,Y 130.322,Z 350.154,A -85,B 0,C 180,E1 -25972.161,E2 -25972.161} C_VEL
LIN {X 0,Y 128.769,Z 363.219,A -85,B 0,C 180,E1 -25973.59,E2 -25973.59} C_VEL
LIN {X 0,Y 126.689,Z 374.778,A -85,B 0,C 180,E1 -25975.345,E2 -25975.345} C_VEL
LIN {X 0,Y 124.228,Z 386.178,A -85,B 0,C 180,E1 -25977.681,E2 -25977.681} C_VEL
LIN {X 0,Y 121.339,Z 398.159,A -85,B 0,C 180,E1 -25980.953,E2 -25980.953} C_VEL
LIN {X 0,Y 118.732,Z 408.395,A -85,B 0,C 180,E1 -25984.586,E2 -25984.586} C_VEL
LIN {X 0,Y 116.412,Z 417.551,A -85,B 0,C 180,E1 -25988.762,E2 -25988.762} C_VEL
LIN {X 0,Y 114.59,Z 426.51,A -85,B 0,C 180,E1 -25993.978,E2 -25993.978} C_VEL
LIN {X 0,Y 113.51,Z 433.624,A -85,B 0,C 180,E1 -25999.294,E2 -25999.294} C_VEL
LIN {X 0,Y 113.432,Z 439.735,A -85,B 0,C 180,E1 -26005.208,E2 -26005.208} C_VEL
LIN {X 0,Y 113.727,Z 443.532,A -85,B 0,C 180,E1 -26009.999,E2 -26009.999} C_VEL
LIN {X 0,Y 113.038,Z 446.619,A -85,B 0,C 180,E1 -26015.851,E2 -26015.851} C_VEL
LIN {X 0,Y 113.05,Z 448.319,A -85,B 0,C 180,E1 -26020.748,E2 -26020.748} C_VEL
LIN {X 0,Y 114.593,Z 449.575,A -85,B 0,C 180,E1 -26027.856,E2 -26027.856} C_VEL
LIN {X 0,Y 118.108,Z 449.418,A -85,B 0,C 180,E1 -26034.615,E2 -26034.615} C_VEL
LIN {X 0,Y 123.171,Z 447.871,A -85,B 0,C 180,E1 -26040.898,E2 -26040.898} C_VEL
LIN {X 0,Y 126.286,Z 446.57,A -85,B 0,C 180,E1 -26043.814,E2 -26043.814} C_VEL
LIN {X 0,Y 133.697,Z 442.81,A -85,B 0,C 180,E1 -26049.108,E2 -26049.108} C_VEL
LIN {X 0,Y 142.409,Z 437.497,A -85,B 0,C 180,E1 -26053.701,E2 -26053.701} C_VEL
LIN {X 0,Y 150.791,Z 431.339,A -85,B 0,C 180,E1 -26057.228,E2 -26057.228} C_VEL
LIN {X 0,Y 159.86,Z 423.559,A -85,B 0,C 180,E1 -26060.295,E2 -26060.295} C_VEL
LIN {X 0,Y 168.087,Z 415.368,A -85,B 0,C 180,E1 -26062.6,E2 -26062.6} C_VEL
LIN {X 0,Y 175.213,Z 407.133,A -85,B 0,C 180,E1 -26064.315,E2 -26064.315} C_VEL
LIN {X 0,Y 180.21,Z 400.593,A -85,B 0,C 180,E1 -26065.351,E2 -26065.351} C_VEL
LIN {X 0,Y 183.199,Z 396.146,A -85,B 0,C 180,E1 -26066.129,E2 -26066.129} C_VEL
LIN {X 0,Y 187.278,Z 388.916,A -85,B 0,C 180,E1 -26067.807,E2 -26067.807} C_VEL
LIN {X 0,Y 191.031,Z 381.357,A -85,B 0,C 180,E1 -26069.368,E2 -26069.368} C_VEL
LIN {X 0,Y 193.426,Z 376.372,A -85,B 0,C 180,E1 -26069.973,E2 -26069.973} C_VEL
LIN {X 0,Y 198.925,Z 363.859,A -85,B 0,C 180,E1 -26070.709,E2 -26070.709} C_VEL
LIN {X 0,Y 203.336,Z 350.699,A -85,B 0,C 180,E1 -26071.286,E2 -26071.286} C_VEL
LIN {X 0,Y 204.08,Z 347.911,A -85,B 0,C 180,E1 -26071.421,E2 -26071.421} C_VEL
LIN {X 0,Y 204.169,Z 346.081,A -85,B 0,C 180,E1 -26073.279,E2 -26073.279} C_VEL
LIN {X 0,Y 204.251,Z 345.078,A -85,B 0,C 180,E1 -26074.896,E2 -26074.896} C_VEL
LIN {X 0,Y 204.676,Z 344.823,A -85,B 0,C 180,E1 -26077.734,E2 -26077.734} C_VEL
LIN {X 0,Y 201.071,Z 356.724,A -85,B 0,C 180,E1 -26078.432,E2 -26078.432} C_VEL
LIN {X 0,Y 195.718,Z 369.927,A -85,B 0,C 180,E1 -26079.468,E2 -26079.468} C_VEL
LIN {X 0,Y 189.247,Z 382.195,A -85,B 0,C 180,E1 -26080.76,E2 -26080.76} C_VEL
LIN {X 0,Y 181.976,Z 393.261,A -85,B 0,C 180,E1 -26082.294,E2 -26082.294} C_VEL
LIN {X 0,Y 174.05,Z 403.091,A -85,B 0,C 180,E1 -26084.182,E2 -26084.182} C_VEL
LIN {X 0,Y 166.449,Z 411.014,A -85,B 0,C 180,E1 -26086.197,E2 -26086.197} C_VEL
LIN {X 0,Y 159.782,Z 416.994,A -85,B 0,C 180,E1 -26088.157,E2 -26088.157} C_VEL
LIN {X 0,Y 150.656,Z 423.915,A -85,B 0,C 180,E1 -26091.28,E2 -26091.28} C_VEL
LIN {X 0,Y 143.054,Z 428.629,A -85,B 0,C 180,E1 -26094.361,E2 -26094.361} C_VEL
LIN {X 0,Y 137.35,Z 431.58,A -85,B 0,C 180,E1 -26097.067,E2 -26097.067} C_VEL
LIN {X 0,Y 131.984,Z 433.928,A -85,B 0,C 180,E1 -26100,E2 -26100} C_VEL
LIN {X 0,Y 126.722,Z 435.701,A -85,B 0,C 180,E1 -26103.376,E2 -26103.376} C_VEL
LIN {X 0,Y 120.683,Z 437.026,A -85,B 0,C 180,E1 -26108.115,E2 -26108.115} C_VEL
LIN {X 0,Y 114.801,Z 437.266,A -85,B 0,C 180,E1 -26114.174,E2 -26114.174} C_VEL
LIN {X 0,Y 111.419,Z 436.532,A -85,B 0,C 180,E1 -26118.891,E2 -26118.891} C_VEL
LIN {X 0,Y 108.385,Z 434.722,A -85,B 0,C 180,E1 -26124.799,E2 -26124.799} C_VEL
LIN {X 0,Y 106.186,Z 431.274,A -85,B 0,C 180,E1 -26131.97,E2 -26131.97} C_VEL
LIN {X 0,Y 105.475,Z 426.224,A -85,B 0,C 180,E1 -26139.269,E2 -26139.269} C_VEL
LIN {X 0,Y 106.058,Z 420.33,A -85,B 0,C 180,E1 -26145.695,E2 -26145.695} C_VEL
LIN {X 0,Y 107.424,Z 413.146,A -85,B 0,C 180,E1 -26151.727,E2 -26151.727} C_VEL
LIN {X 0,Y 109.469,Z 404.433,A -85,B 0,C 180,E1 -26157.439,E2 -26157.439} C_VEL
LIN {X 0,Y 112.041,Z 394.692,A -85,B 0,C 180,E1 -26162.404,E2 -26162.404} C_VEL
LIN {X 0,Y 114.849,Z 383.996,A -85,B 0,C 180,E1 -26166.62,E2 -26166.62} C_VEL
LIN {X 0,Y 117.69,Z 372.279,A -85,B 0,C 180,E1 -26170.177,E2 -26170.177} C_VEL
LIN {X 0,Y 120.346,Z 359.797,A -85,B 0,C 180,E1 -26173.024,E2 -26173.024} C_VEL
LIN {X 0,Y 122.517,Z 347.629,A -85,B 0,C 180,E1 -26175.09,E2 -26175.09} C_VEL
LIN {X 0,Y 124.242,Z 333.894,A -85,B 0,C 180,E1 -26176.731,E2 -26176.731} C_VEL
LIN {X 0,Y 126.128,Z 310.317,A -85,B 0,C 180,E1 -26178.457,E2 -26178.457} C_VEL
LIN {X 0,Y 128.246,Z 286.127,A -85,B 0,C 180,E1 -26180,E2 -26180} C_VEL
LIN {X 0,Y 121.766,Z 269.23,A -85,B 0,C 180,E1 -26183.054,E2 -26183.054} C_VEL
LIN {X 0,Y 115.582,Z 255.289,A -85,B 0,C 180,E1 -26186.069,E2 -26186.069} C_VEL
LIN {X 0,Y 109.049,Z 241.967,A -85,B 0,C 180,E1 -26189.598,E2 -26189.598} C_VEL
LIN {X 0,Y 108.912,Z 240.917,A -85,B 0,C 180,E1 -26189.886,E2 -26189.886} C_VEL
LIN {X 0,Y 108.3,Z 240.993,A -85,B 0,C 180,E1 -26197.458,E2 -26197.458} C_VEL
LIN {X 0,Y 108.174,Z 241.01,A -85,B 0,C 180,E1 -26202.956,E2 -26202.956} C_VEL
LIN {X 0,Y 107.905,Z 241.031,A -85,B 0,C 180,E1 -26209.007,E2 -26209.007} C_VEL
LIN {X 0,Y 107.856,Z 241.033,A -85,B 0,C 180,E1 -26214.182,E2 -26214.182} C_VEL
LIN {X 0,Y 107.779,Z 241.052,A -85,B 0,C 180,E1 -26222.038,E2 -26222.038} C_VEL
LIN {X 0,Y 107.682,Z 241.026,A -85,B 0,C 180,E1 -26228.446,E2 -26228.446} C_VEL
LIN {X 0,Y 107.671,Z 241.071,A -85,B 0,C 180,E1 -26235.891,E2 -26235.891} C_VEL
LIN {X 0,Y 107.684,Z 241.061,A -85,B 0,C 180,E1 -26241.554,E2 -26241.554} C_VEL
LIN {X 0,Y 107.793,Z 241.057,A -85,B 0,C 180,E1 -26248.561,E2 -26248.561} C_VEL
LIN {X 0,Y 107.912,Z 241.035,A -85,B 0,C 180,E1 -26256.998,E2 -26256.998} C_VEL
LIN {X 0,Y 108.017,Z 241.014,A -85,B 0,C 180,E1 -26264.915,E2 -26264.915} C_VEL
LIN {X 0,Y 108.21,Z 240.96,A -85,B 0,C 180,E1 -26268.765,E2 -26268.765} C_VEL
LIN {X 0,Y 108.293,Z 240.956,A -85,B 0,C 180,E1 -26272.542,E2 -26272.542} C_VEL
LIN {X 0,Y 108.902,Z 240.92,A -85,B 0,C 180,E1 -26280,E2 -26280} C_VEL
LIN {X 0,Y 108.29,Z 240.964,A -85,B 0,C 180,E1 -26287.458,E2 -26287.458} C_VEL
LIN {X 0,Y 108.141,Z 241.012,A -85,B 0,C 180,E1 -26292.874,E2 -26292.874} C_VEL
LIN {X 0,Y 107.866,Z 241.039,A -85,B 0,C 180,E1 -26299.013,E2 -26299.013} C_VEL
LIN {X 0,Y 107.819,Z 241.053,A -85,B 0,C 180,E1 -26304.135,E2 -26304.135} C_VEL
LIN {X 0,Y 107.78,Z 241.052,A -85,B 0,C 180,E1 -26312.037,E2 -26312.037} C_VEL
LIN {X 0,Y 107.745,Z 241.247,A -85,B 0,C 180,E1 -26316.361,E2 -26316.361} C_VEL
LIN {X 0,Y 108.949,Z 244.215,A -85,B 0,C 180,E1 -26317.126,E2 -26317.126} C_VEL
LIN {X 0,Y 112.768,Z 250.922,A -85,B 0,C 180,E1 -26319.126,E2 -26319.126} C_VEL
LIN {X 0,Y 118.374,Z 265.375,A -85,B 0,C 180,E1 -26322.194,E2 -26322.194} C_VEL
LIN {X 0,Y 123.889,Z 282.207,A -85,B 0,C 180,E1 -26325.162,E2 -26325.162} C_VEL
LIN {X 0,Y 124.997,Z 286.49,A -85,B 0,C 180,E1 -26325.797,E2 -26325.797} C_VEL
LIN {X 0,Y 126.509,Z 316.347,A -85,B 0,C 180,E1 -26328.644,E2 -26328.644} C_VEL
LIN {X 0,Y 123.671,Z 350.458,A -85,B 0,C 180,E1 -26331.047,E2 -26331.047} C_VEL
LIN {X 0,Y 122.042,Z 363.263,A -85,B 0,C 180,E1 -26332.535,E2 -26332.535} C_VEL
LIN {X 0,Y 119.705,Z 375.668,A -85,B 0,C 180,E1 -26334.564,E2 -26334.564} C_VEL
LIN {X 0,Y 116.741,Z 388.693,A -85,B 0,C 180,E1 -26337.53,E2 -26337.53} C_VEL
LIN {X 0,Y 113.871,Z 399.809,A -85,B 0,C 180,E1 -26340.918,E2 -26340.918} C_VEL
LIN {X 0,Y 111.267,Z 409.523,A -85,B 0,C 180,E1 -26344.763,E2 -26344.763} C_VEL
LIN {X 0,Y 109.064,Z 418.427,A -85,B 0,C 180,E1 -26349.241,E2 -26349.241} C_VEL
LIN {X 0,Y 107.32,Z 427.104,A -85,B 0,C 180,E1 -26354.813,E2 -26354.813} C_VEL
LIN {X 0,Y 106.392,Z 433.946,A -85,B 0,C 180,E1 -26360.493,E2 -26360.493} C_VEL
LIN {X 0,Y 106.468,Z 439.354,A -85,B 0,C 180,E1 -26366.214,E2 -26366.214} C_VEL
LIN {X 0,Y 106.711,Z 442.212,A -85,B 0,C 180,E1 -26369.999,E2 -26369.999} C_VEL
LIN {X 0,Y 106.042,Z 445.476,A -85,B 0,C 180,E1 -26376.204,E2 -26376.204} C_VEL
LIN {X 0,Y 106.102,Z 447.329,A -85,B 0,C 180,E1 -26381.461,E2 -26381.461} C_VEL
LIN {X 0,Y 107.848,Z 448.829,A -85,B 0,C 180,E1 -26389.015,E2 -26389.015} C_VEL
LIN {X 0,Y 111.667,Z 448.933,A -85,B 0,C 180,E1 -26396.138,E2 -26396.138} C_VEL
LIN {X 0,Y 117.101,Z 447.603,A -85,B 0,C 180,E1 -26402.693,E2 -26402.693} C_VEL
LIN {X 0,Y 124.182,Z 444.91,A -85,B 0,C 180,E1 -26408.501,E2 -26408.501} C_VEL
LIN {X 0,Y 130.456,Z 441.904,A -85,B 0,C 180,E1 -26412.33,E2 -26412.33} C_VEL
LIN {X 0,Y 139.815,Z 436.493,A -85,B 0,C 180,E1 -26416.79,E2 -26416.79} C_VEL
LIN {X 0,Y 148.733,Z 430.279,A -85,B 0,C 180,E1 -26420.16,E2 -26420.16} C_VEL
LIN {X 0,Y 158.258,Z 422.437,A -85,B 0,C 180,E1 -26423.067,E2 -26423.067} C_VEL
LIN {X 0,Y 166.857,Z 414.117,A -85,B 0,C 180,E1 -26425.218,E2 -26425.218} C_VEL
LIN {X 0,Y 174.251,Z 405.833,A -85,B 0,C 180,E1 -26426.814,E2 -26426.814} C_VEL
LIN {X 0,Y 182.695,Z 394.643,A -85,B 0,C 180,E1 -26428.332,E2 -26428.332} C_VEL
LIN {X 0,Y 189.769,Z 383.331,A -85,B 0,C 180,E1 -26429.434,E2 -26429.434} C_VEL
LIN {X 0,Y 193.426,Z 376.372,A -85,B 0,C 180,E1 -26429.973,E2 -26429.973} C_VEL
LIN {X 0,Y 194.958,Z 372.986,A -85,B 0,C 180,E1 -26430.417,E2 -26430.417} C_VEL
LIN {X 0,Y 198.861,Z 362.56,A -85,B 0,C 180,E1 -26432.637,E2 -26432.637} C_VEL
LIN {X 0,Y 200.129,Z 359.001,A -85,B 0,C 180,E1 -26432.986,E2 -26432.986} C_VEL
LIN {X 0,Y 201.74,Z 354.295,A -85,B 0,C 180,E1 -26433.167,E2 -26433.167} C_VEL
LIN {X 0,Y 202.159,Z 352.703,A -85,B 0,C 180,E1 -26433.731,E2 -26433.731} C_VEL
LIN {X 0,Y 202.334,Z 351.767,A -85,B 0,C 180,E1 -26435.366,E2 -26435.366} C_VEL
LIN {X 0,Y 202.404,Z 351.649,A -85,B 0,C 180,E1 -26435.858,E2 -26435.858} C_VEL
LIN {X 0,Y 202.292,Z 352.056,A -85,B 0,C 180,E1 -26436.084,E2 -26436.084} C_VEL
LIN {X 0,Y 197.496,Z 365.08,A -85,B 0,C 180,E1 -26436.956,E2 -26436.956} C_VEL
LIN {X 0,Y 191.912,Z 376.577,A -85,B 0,C 180,E1 -26437.953,E2 -26437.953} C_VEL
LIN {X 0,Y 185.29,Z 387.479,A -85,B 0,C 180,E1 -26439.169,E2 -26439.169} C_VEL
LIN {X 0,Y 177.714,Z 397.779,A -85,B 0,C 180,E1 -26440.7,E2 -26440.7} C_VEL
LIN {X 0,Y 169.43,Z 407.045,A -85,B 0,C 180,E1 -26442.561,E2 -26442.561} C_VEL
LIN {X 0,Y 160.125,Z 415.655,A -85,B 0,C 180,E1 -26444.925,E2 -26444.925} C_VEL
LIN {X 0,Y 151.104,Z 422.506,A -85,B 0,C 180,E1 -26447.612,E2 -26447.612} C_VEL
LIN {X 0,Y 142.445,Z 427.949,A -85,B 0,C 180,E1 -26450.665,E2 -26450.665} C_VEL
LIN {X 0,Y 134.237,Z 432.108,A -85,B 0,C 180,E1 -26454.12,E2 -26454.12} C_VEL
LIN {X 0,Y 126.577,Z 435.098,A -85,B 0,C 180,E1 -26458.028,E2 -26458.028} C_VEL
LIN {X 0,Y 118.31,Z 437.299,A -85,B 0,C 180,E1 -26463.405,E2 -26463.405} C_VEL
LIN {X 0,Y 113.402,Z 437.888,A -85,B 0,C 180,E1 -26467.443,E2 -26467.443} C_VEL
LIN {X 0,Y 108.158,Z 437.715,A -85,B 0,C 180,E1 -26472.923,E2 -26472.923} C_VEL
LIN {X 0,Y 103.434,Z 436.243,A -85,B 0,C 180,E1 -26479.86,E2 -26479.86} C_VEL
LIN {X 0,Y 100.245,Z 433.349,A -85,B 0,C 180,E1 -26487.239,E2 -26487.239} C_VEL
LIN {X 0,Y 98.616,Z 429.094,A -85,B 0,C 180,E1 -26494.759,E2 -26494.759} C_VEL
LIN {X 0,Y 98.533,Z 423.359,A -85,B 0,C 180,E1 -26502.32,E2 -26502.32} C_VEL
LIN {X 0,Y 99.371,Z 417.827,A -85,B 0,C 180,E1 -26507.954,E2 -26507.954} C_VEL
LIN {X 0,Y 100.738,Z 411.267,A -85,B 0,C 180,E1 -26513.346,E2 -26513.346} C_VEL
LIN {X 0,Y 102.801,Z 402.946,A -85,B 0,C 180,E1 -26518.799,E2 -26518.799} C_VEL
LIN {X 0,Y 105.349,Z 393.684,A -85,B 0,C 180,E1 -26523.591,E2 -26523.591} C_VEL
LIN {X 0,Y 108.382,Z 382.471,A -85,B 0,C 180,E1 -26528.11,E2 -26528.11} C_VEL
LIN {X 0,Y 111.425,Z 370.395,A -85,B 0,C 180,E1 -26531.774,E2 -26531.774} C_VEL
LIN {X 0,Y 114.051,Z 358.166,A -85,B 0,C 180,E1 -26534.59,E2 -26534.59} C_VEL
LIN {X 0,Y 116.289,Z 345.588,A -85,B 0,C 180,E1 -26536.686,E2 -26536.686} C_VEL
LIN {X 0,Y 117.928,Z 332.105,A -85,B 0,C 180,E1 -26538.28,E2 -26538.28} C_VEL
LIN {X 0,Y 121.781,Z 287.361,A -85,B 0,C 180,E1 -26541.441,E2 -26541.441} C_VEL
LIN {X 0,Y 115.504,Z 271.369,A -85,B 0,C 180,E1 -26544.547,E2 -26544.547} C_VEL
LIN {X 0,Y 110.156,Z 259.004,A -85,B 0,C 180,E1 -26547.43,E2 -26547.43} C_VEL
LIN {X 0,Y 103.534,Z 245.804,A -85,B 0,C 180,E1 -26551.255,E2 -26551.255} C_VEL
LIN {X 0,Y 101.858,Z 243.239,A -85,B 0,C 180,E1 -26552.224,E2 -26552.224} C_VEL
LIN {X 0,Y 101.5,Z 241.839,A -85,B 0,C 180,E1 -26552.604,E2 -26552.604} C_VEL
LIN {X 0,Y 101.24,Z 241.873,A -85,B 0,C 180,E1 -26557.982,E2 -26557.982} C_VEL
LIN {X 0,Y 101.103,Z 241.891,A -85,B 0,C 180,E1 -26563.298,E2 -26563.298} C_VEL
LIN {X 0,Y 100.817,Z 241.903,A -85,B 0,C 180,E1 -26570.4,E2 -26570.4} C_VEL
LIN {X 0,Y 100.776,Z 241.919,A -85,B 0,C 180,E1 -26574.96,E2 -26574.96} C_VEL
LIN {X 0,Y 100.688,Z 241.927,A -85,B 0,C 180,E1 -26583.113,E2 -26583.113} C_VEL
LIN {X 0,Y 100.634,Z 241.909,A -85,B 0,C 180,E1 -26589.807,E2 -26589.807} C_VEL
LIN {X 0,Y 100.642,Z 241.946,A -85,B 0,C 180,E1 -26595.708,E2 -26595.708} C_VEL
LIN {X 0,Y 100.622,Z 241.942,A -85,B 0,C 180,E1 -26601.053,E2 -26601.053} C_VEL
LIN {X 0,Y 100.689,Z 241.94,A -85,B 0,C 180,E1 -26606.888,E2 -26606.888} C_VEL
LIN {X 0,Y 100.788,Z 241.916,A -85,B 0,C 180,E1 -26615.268,E2 -26615.268} C_VEL
LIN {X 0,Y 100.815,Z 241.925,A -85,B 0,C 180,E1 -26619.601,E2 -26619.601} C_VEL
LIN {X 0,Y 101.119,Z 241.847,A -85,B 0,C 180,E1 -26627.965,E2 -26627.965} C_VEL
LIN {X 0,Y 101.227,Z 241.83,A -85,B 0,C 180,E1 -26632.019,E2 -26632.019} C_VEL
LIN {X 0,Y 101.83,Z 241.801,A -85,B 0,C 180,E1 -26640,E2 -26640} C_VEL
LIN {X 0,Y 101.224,Z 241.843,A -85,B 0,C 180,E1 -26647.982,E2 -26647.982} C_VEL
LIN {X 0,Y 101.053,Z 241.896,A -85,B 0,C 180,E1 -26653.173,E2 -26653.173} C_VEL
LIN {X 0,Y 100.782,Z 241.914,A -85,B 0,C 180,E1 -26660.407,E2 -26660.407} C_VEL
LIN {X 0,Y 100.736,Z 241.939,A -85,B 0,C 180,E1 -26664.908,E2 -26664.908} C_VEL
LIN {X 0,Y 100.684,Z 241.942,A -85,B 0,C 180,E1 -26673.107,E2 -26673.107} C_VEL
LIN {X 0,Y 100.671,Z 242.077,A -85,B 0,C 180,E1 -26673.636,E2 -26673.636} C_VEL
LIN {X 0,Y 101.763,Z 244.944,A -85,B 0,C 180,E1 -26674.433,E2 -26674.433} C_VEL
LIN {X 0,Y 103.196,Z 247.121,A -85,B 0,C 180,E1 -26675.262,E2 -26675.262} C_VEL
LIN {X 0,Y 107.739,Z 255.501,A -85,B 0,C 180,E1 -26677.895,E2 -26677.895} C_VEL
LIN {X 0,Y 113.041,Z 269.666,A -85,B 0,C 180,E1 -26681.067,E2 -26681.067} C_VEL
LIN {X 0,Y 118.688,Z 287.496,A -85,B 0,C 180,E1 -26684.311,E2 -26684.311} C_VEL
LIN {X 0,Y 120.078,Z 316.336,A -85,B 0,C 180,E1 -26687.251,E2 -26687.251} C_VEL
LIN {X 0,Y 117.167,Z 349.771,A -85,B 0,C 180,E1 -26689.706,E2 -26689.706} C_VEL
LIN {X 0,Y 115.371,Z 363.315,A -85,B 0,C 180,E1 -26691.361,E2 -26691.361} C_VEL
LIN {X 0,Y 112.755,Z 376.493,A -85,B 0,C 180,E1 -26693.69,E2 -26693.69} C_VEL
LIN {X 0,Y 109.979,Z 388.076,A -85,B 0,C 180,E1 -26696.494,E2 -26696.494} C_VEL
LIN {X 0,Y 107.067,Z 398.938,A -85,B 0,C 180,E1 -26699.965,E2 -26699.965} C_VEL
LIN {X 0,Y 104.358,Z 408.672,A -85,B 0,C 180,E1 -26704.039,E2 -26704.039} C_VEL
LIN {X 0,Y 102.059,Z 417.588,A -85,B 0,C 180,E1 -26708.805,E2 -26708.805} C_VEL
